C03618=1103.149,283.169,-77.538,179.285,15.809,151.491
C03619=1103.143,282.921,-77.509,179.281,15.808,151.491
C03620=1103.138,282.672,-77.480,179.278,15.807,151.492
C03621=1103.132,282.424,-77.450,179.274,15.805,151.492
C03622=1103.126,282.176,-77.422,179.271,15.805,151.493
C03623=1103.121,281.927,-77.393,179.267,15.803,151.493
C03624=1103.115,281.679,-77.364,179.264,15.802,151.494
C03625=1103.109,281.431,-77.334,179.260,15.801,151.494
C03626=1103.104,281.183,-77.305,179.256,15.800,151.495
C03627=1103.098,280.935,-77.276,179.252,15.799,151.495
C03628=1103.092,280.687,-77.247,179.249,15.798,151.496
C03629=1103.087,280.438,-77.218,179.245,15.797,151.496
C03630=1103.081,280.190,-77.189,179.242,15.796,151.497
C03631=1103.076,279.942,-77.159,179.238,15.795,151.497
C03632=1103.069,279.694,-77.130,179.235,15.794,151.498
C03633=1103.064,279.446,-77.101,179.231,15.793,151.498
C03634=1103.059,279.197,-77.073,179.227,15.792,151.499
C03635=1103.053,278.949,-77.043,179.224,15.791,151.499
C03636=1103.047,278.701,-77.014,179.220,15.790,151.500
C03637=1103.041,278.453,-76.986,179.216,15.789,151.500
C03638=1103.036,278.204,-76.956,179.212,15.788,151.501
C03639=1103.030,277.956,-76.927,179.209,15.787,151.502
C03640=1103.025,277.708,-76.899,179.205,15.786,151.502
C03641=1103.019,277.460,-76.870,179.202,15.785,151.503
C03642=1103.013,277.211,-76.841,179.198,15.784,151.503
C03643=1103.008,276.963,-76.812,179.195,15.783,151.504
C03644=1103.000,276.606,-76.771,179.189,15.782,151.504
C03645=1102.991,276.250,-76.729,179.184,15.781,151.505
C03646=1102.984,275.893,-76.688,179.179,15.780,151.506
C03647=1102.975,275.536,-76.647,179.174,15.778,151.507
C03648=1102.969,275.288,-76.618,179.170,15.777,151.507
C03649=1102.964,275.039,-76.589,179.167,15.776,151.508
C03650=1102.958,274.791,-76.560,179.163,15.775,151.508
C03651=1102.952,274.543,-76.532,179.159,15.774,151.509
C03652=1102.946,274.294,-76.503,179.155,15.773,151.509
C03653=1102.941,274.046,-76.474,179.152,15.772,151.510
C03654=1102.935,273.797,-76.446,179.148,15.771,151.511
C03655=1102.930,273.550,-76.417,179.145,15.770,151.511
C03656=1102.924,273.301,-76.389,179.141,15.769,151.512
C03657=1102.918,273.053,-76.359,179.138,15.769,151.512
C03658=1102.913,272.805,-76.331,179.134,15.767,151.513
C03659=1102.907,272.556,-76.303,179.130,15.767,151.513
C03660=1102.901,272.308,-76.274,179.127,15.766,151.514
C03661=1102.896,272.060,-76.246,179.123,15.765,151.515
C03662=1102.891,271.811,-76.217,179.120,15.764,151.515
C03663=1102.885,271.563,-76.188,179.116,15.763,151.516
C03664=1102.879,271.314,-76.160,179.112,15.762,151.516
C03665=1102.873,271.066,-76.132,179.108,15.762,151.517
C03666=1102.867,270.818,-76.103,179.105,15.761,151.517
C03667=1102.862,270.570,-76.075,179.101,15.760,151.518
C03668=1102.856,270.321,-76.047,179.098,15.759,151.518
C03669=1102.851,270.073,-76.019,179.094,15.758,151.519
C03670=1102.845,269.825,-75.989,179.090,15.757,151.520
C03671=1102.840,269.577,-75.961,179.086,15.756,151.520
C03672=1102.834,269.328,-75.933,179.083,15.756,151.521
C03673=1102.828,269.079,-75.904,179.080,15.755,151.521
C03674=1102.822,268.831,-75.876,179.076,15.754,151.522
C03675=1102.816,268.583,-75.848,179.072,15.753,151.522
C03676=1102.811,268.335,-75.819,179.068,15.752,151.523
C03677=1102.805,268.086,-75.791,179.065,15.751,151.524
C03678=1102.800,267.838,-75.763,179.061,15.750,151.524
C03679=1102.794,267.590,-75.735,179.057,15.750,151.525
C03680=1102.788,267.342,-75.707,179.054,15.749,151.525
C03681=1102.782,267.093,-75.679,179.050,15.748,151.526
C03682=1102.777,266.845,-75.651,179.047,15.748,151.527
C03683=1102.771,266.596,-75.622,179.043,15.746,151.527
C03684=1102.766,266.348,-75.594,179.040,15.746,151.528
C03685=1102.760,266.100,-75.566,179.035,15.745,151.528
C03686=1102.754,265.851,-75.538,179.032,15.744,151.529
C03687=1102.749,265.603,-75.510,179.028,15.743,151.529
C03688=1102.743,265.354,-75.482,179.025,15.743,151.530
C03689=1102.738,265.106,-75.454,179.021,15.742,151.531
C03690=1102.732,264.858,-75.425,179.017,15.741,151.531
C03691=1102.726,264.610,-75.398,179.014,15.740,151.532
C03692=1102.720,264.362,-75.370,179.010,15.739,151.532
C03693=1102.714,264.113,-75.342,179.006,15.739,151.533
C03694=1102.709,263.865,-75.314,179.003,15.738,151.534
C03695=1102.703,263.616,-75.286,178.999,15.737,151.534
C03696=1102.695,263.263,-75.246,178.994,15.736,151.535
C03697=1102.686,262.908,-75.207,178.988,15.735,151.536
C03698=1102.679,262.554,-75.167,178.984,15.735,151.537
C03699=1102.670,262.200,-75.127,178.978,15.733,151.538
C03700=1102.665,261.952,-75.099,178.974,15.732,151.538
C03701=1102.659,261.703,-75.071,178.971,15.732,151.539
C03702=1102.653,261.455,-75.044,178.968,15.731,151.539
C03703=1102.647,261.206,-75.016,178.963,15.730,151.540
C03704=1102.642,260.958,-74.988,178.960,15.730,151.541
C03705=1102.636,260.710,-74.960,178.956,15.729,151.541
C03706=1102.630,260.461,-74.933,178.953,15.728,151.542
C03707=1102.625,260.213,-74.905,178.949,15.728,151.543
C03708=1102.618,259.964,-74.877,178.945,15.727,151.543
C03709=1102.613,259.716,-74.850,178.941,15.726,151.544
C03710=1102.608,259.468,-74.822,178.938,15.726,151.544
C03711=1102.601,259.219,-74.794,178.934,15.725,151.545
C03712=1102.596,258.971,-74.767,178.931,15.724,151.546
C03713=1102.591,258.723,-74.739,178.926,15.723,151.546
C03714=1102.584,258.474,-74.711,178.923,15.723,151.547
C03715=1102.579,258.225,-74.684,178.920,15.722,151.548
C03716=1102.573,257.977,-74.656,178.915,15.721,151.548
C03717=1102.567,257.728,-74.629,178.912,15.721,151.549
C03718=1102.562,257.480,-74.601,178.909,15.721,151.549
C03719=1102.556,257.233,-74.574,178.905,15.719,151.550
C03720=1102.550,256.983,-74.546,178.901,15.719,151.551
C03721=1102.545,256.735,-74.518,178.898,15.718,151.551
C03722=1102.539,256.487,-74.491,178.894,15.717,151.552
C03723=1102.533,256.238,-74.463,178.890,15.717,151.552
C03724=1102.527,255.990,-74.436,178.886,15.716,151.553
C03725=1102.522,255.742,-74.409,178.883,15.715,151.554
C03726=1102.517,255.493,-74.381,178.879,15.715,151.554
C03727=1102.510,255.244,-74.354,178.875,15.714,151.555
C03728=1102.505,254.996,-74.326,178.872,15.714,151.556
C03729=1102.499,254.747,-74.300,178.868,15.713,151.556
C03730=1102.494,254.499,-74.272,178.864,15.712,151.557
C03731=1102.488,254.250,-74.245,178.861,15.712,151.558
C03732=1102.483,254.002,-74.217,178.858,15.711,151.558
C03733=1102.476,253.754,-74.190,178.853,15.710,151.559
C03734=1102.471,253.505,-74.163,178.850,15.710,151.559
C03735=1102.465,253.257,-74.135,178.847,15.709,151.560
C03736=1102.460,253.008,-74.108,178.843,15.708,151.561
C03737=1102.454,252.760,-74.081,178.839,15.708,151.561
C03738=1102.449,252.511,-74.054,178.835,15.707,151.562
C03739=1102.443,252.263,-74.027,178.832,15.706,151.562
C03740=1102.438,252.015,-73.999,178.828,15.706,151.563
C03741=1102.431,251.766,-73.972,178.824,15.705,151.564
C03742=1102.426,251.517,-73.945,178.821,15.705,151.564
C03743=1102.420,251.269,-73.918,178.817,15.704,151.565
C03744=1102.415,251.021,-73.891,178.813,15.703,151.566
C03745=1102.410,250.772,-73.864,178.810,15.702,151.566
C03746=1102.404,250.524,-73.837,178.806,15.702,151.567
C03747=1102.398,250.274,-73.810,178.802,15.701,151.568
C03748=1102.390,249.918,-73.770,178.797,15.701,151.568
C03749=1102.382,249.561,-73.732,178.792,15.700,151.569
C03750=1102.374,249.204,-73.693,178.787,15.699,151.570
C03751=1102.366,248.847,-73.653,178.781,15.698,151.571
C03752=1102.361,248.599,-73.627,178.778,15.697,151.572
C03753=1102.355,248.351,-73.600,178.775,15.697,151.572
C03754=1102.350,248.102,-73.573,178.770,15.696,151.573
C03755=1102.344,247.854,-73.546,178.767,15.695,151.574
C03756=1102.339,247.605,-73.519,178.764,15.695,151.574
C03757=1102.333,247.357,-73.492,178.760,15.694,151.575
C03758=1102.327,247.108,-73.466,178.756,15.694,151.575
C03759=1102.322,246.860,-73.439,178.753,15.693,151.576
C03760=1102.317,246.611,-73.412,178.749,15.692,151.577
C03761=1102.311,246.363,-73.385,178.745,15.692,151.577
C03762=1102.304,246.114,-73.358,178.741,15.692,151.578
C03763=1102.299,245.865,-73.332,178.738,15.691,151.579
C03764=1102.294,245.617,-73.304,178.734,15.690,151.579
C03765=1102.288,245.368,-73.278,178.730,15.690,151.580
C03766=1102.282,245.120,-73.251,178.727,15.689,151.581
C03767=1102.276,244.872,-73.224,178.723,15.688,151.581
C03768=1102.272,244.622,-73.198,178.719,15.688,151.582
C03769=1102.266,244.374,-73.171,178.716,15.688,151.583
C03770=1102.260,244.126,-73.145,178.713,15.687,151.583
C03771=1102.254,243.877,-73.118,178.708,15.687,151.584
C03772=1102.248,243.629,-73.091,178.705,15.686,151.584
C03773=1102.243,243.381,-73.065,178.702,15.686,151.585
C03774=1102.238,243.131,-73.038,178.697,15.685,151.586
C03775=1102.232,242.883,-73.011,178.694,15.684,151.586
C03776=1102.226,242.635,-72.985,178.691,15.684,151.587
C03777=1102.221,242.386,-72.958,178.687,15.684,151.588
C03778=1102.215,242.138,-72.931,178.683,15.683,151.589
C03779=1102.209,241.889,-72.906,178.680,15.682,151.589
C03780=1102.204,241.641,-72.879,178.676,15.682,151.590
C03781=1102.198,241.392,-72.852,178.672,15.681,151.590
C03782=1102.192,241.144,-72.826,178.668,15.681,151.591
C03783=1102.187,240.895,-72.800,178.665,15.681,151.592
C03784=1102.181,240.646,-72.773,178.661,15.680,151.592
C03785=1102.175,240.398,-72.746,178.657,15.679,151.593
C03786=1102.170,240.149,-72.720,178.654,15.679,151.594
C03787=1102.164,239.901,-72.694,178.650,15.679,151.595
C03788=1102.158,239.652,-72.667,178.647,15.678,151.595
C03789=1102.153,239.403,-72.641,178.642,15.677,151.596
C03790=1102.147,239.155,-72.615,178.639,15.677,151.597
C03791=1102.141,238.906,-72.589,178.635,15.677,151.597
C03792=1102.136,238.658,-72.562,178.632,15.676,151.598
C03793=1102.130,238.409,-72.535,178.628,15.676,151.598
C03794=1102.124,238.160,-72.509,178.624,15.675,151.599
C03795=1102.119,237.912,-72.483,178.621,15.675,151.600
C03796=1102.113,237.663,-72.457,178.617,15.675,151.601
C03797=1102.107,237.415,-72.431,178.613,15.674,151.601
C03798=1102.101,237.166,-72.405,178.610,15.674,151.602
C03799=1102.095,236.918,-72.378,178.606,15.673,151.603
C03800=1102.088,236.554,-72.340,178.601,15.672,151.603
C03801=1102.079,236.190,-72.302,178.595,15.672,151.604
C03802=1102.071,235.827,-72.263,178.591,15.671,151.605
C03803=1102.063,235.463,-72.226,178.585,15.671,151.606
C03804=1102.057,235.214,-72.199,178.581,15.670,151.607
C03805=1102.052,234.965,-72.173,178.578,15.670,151.608
C03806=1102.046,234.718,-72.147,178.574,15.669,151.608
C03807=1102.041,234.469,-72.121,178.570,15.669,151.609
C03808=1102.035,234.220,-72.095,178.567,15.669,151.610
C03809=1102.029,233.972,-72.069,178.563,15.668,151.610
C03810=1102.023,233.723,-72.043,178.559,15.667,151.611
C03811=1102.018,233.474,-72.017,178.556,15.667,151.612
C03812=1102.013,233.226,-71.991,178.552,15.667,151.612
C03813=1102.007,232.977,-71.966,178.549,15.667,151.613
C03814=1102.001,232.728,-71.940,178.545,15.666,151.614
C03815=1101.996,232.479,-71.914,178.541,15.666,151.615
C03816=1101.990,232.231,-71.887,178.538,15.665,151.615
C03817=1101.984,231.982,-71.862,178.534,15.665,151.616
C03818=1101.979,231.734,-71.836,178.530,15.665,151.617
C03819=1101.973,231.485,-71.810,178.526,15.664,151.617
C03820=1101.968,231.237,-71.784,178.523,15.663,151.618
C03821=1101.961,230.988,-71.758,178.519,15.663,151.619
C03822=1101.956,230.739,-71.732,178.516,15.663,151.619
C03823=1101.951,230.491,-71.707,178.512,15.662,151.620
C03824=1101.945,230.242,-71.681,178.508,15.662,151.621
C03825=1101.939,229.993,-71.655,178.505,15.661,151.621
C03826=1101.933,229.745,-71.629,178.501,15.661,151.622
C03827=1101.927,229.496,-71.603,178.497,15.661,151.623
C03828=1101.923,229.248,-71.578,178.494,15.661,151.623
C03829=1101.916,228.999,-71.553,178.491,15.660,151.624
C03830=1101.911,228.750,-71.527,178.486,15.659,151.625
C03831=1101.905,228.502,-71.501,178.483,15.659,151.625
C03832=1101.900,228.253,-71.476,178.479,15.659,151.626
C03833=1101.894,228.005,-71.450,178.476,15.659,151.627
C03834=1101.888,227.756,-71.424,178.472,15.659,151.628
C03835=1101.882,227.507,-71.399,178.468,15.658,151.628
C03836=1101.877,227.259,-71.374,178.464,15.658,151.629
C03837=1101.872,227.010,-71.348,178.461,15.658,151.630
C03838=1101.865,226.761,-71.322,178.458,15.657,151.630
C03839=1101.860,226.512,-71.296,178.454,15.657,151.631
C03840=1101.854,226.264,-71.271,178.451,15.657,151.632
C03841=1101.849,226.015,-71.245,178.446,15.656,151.632
C03842=1101.843,225.766,-71.220,178.443,15.656,151.633
C03843=1101.838,225.518,-71.194,178.439,15.655,151.634
C03844=1101.832,225.269,-71.169,178.436,15.655,151.635
C03845=1101.826,225.020,-71.143,178.432,15.655,151.635
C03846=1101.820,224.772,-71.118,178.429,15.654,151.636
C03847=1101.815,224.523,-71.094,178.425,15.654,151.636
C03848=1101.809,224.274,-71.068,178.421,15.653,151.637
C03849=1101.803,224.026,-71.042,178.417,15.653,151.638
C03850=1101.798,223.777,-71.017,178.414,15.653,151.639
C03851=1101.792,223.529,-70.991,178.410,15.653,151.639
C03852=1101.784,223.156,-70.954,178.405,15.652,151.640
C03853=1101.776,222.784,-70.916,178.399,15.651,151.641
C03854=1101.767,222.412,-70.878,178.394,15.651,151.642
C03855=1101.759,222.040,-70.840,178.389,15.651,151.643
C03856=1101.753,221.792,-70.815,178.385,15.651,151.644
C03857=1101.747,221.543,-70.790,178.382,15.650,151.645
C03858=1101.741,221.294,-70.764,178.377,15.650,151.646
C03859=1101.737,221.045,-70.740,178.374,15.649,151.646
C03860=1101.730,220.797,-70.714,178.370,15.649,151.647
C03861=1101.724,220.548,-70.689,178.367,15.649,151.648
C03862=1101.719,220.299,-70.665,178.363,15.649,151.648
C03863=1101.713,220.050,-70.639,178.360,15.649,151.649
C03864=1101.707,219.802,-70.613,178.356,15.649,151.650
C03865=1101.702,219.553,-70.589,178.352,15.648,151.651
C03866=1101.696,219.304,-70.564,178.349,15.647,151.651
C03867=1101.691,219.056,-70.539,178.345,15.647,151.652
C03868=1101.685,218.807,-70.514,178.341,15.647,151.653
C03869=1101.679,218.559,-70.489,178.338,15.647,151.653
C03870=1101.673,218.310,-70.464,178.334,15.647,151.654
C03871=1101.668,218.061,-70.438,178.331,15.646,151.655
C03872=1101.663,217.812,-70.414,178.327,15.646,151.655
C03873=1101.656,217.563,-70.388,178.323,15.645,151.656
C03874=1101.651,217.315,-70.364,178.319,15.645,151.657
C03875=1101.645,217.066,-70.339,178.316,15.645,151.658
C03876=1101.640,216.817,-70.314,178.312,15.645,151.658
C03877=1101.634,216.569,-70.289,178.309,15.645,151.659
C03878=1101.629,216.320,-70.264,178.305,15.645,151.660
C03879=1101.623,216.071,-70.239,178.302,15.644,151.660
C03880=1101.617,215.823,-70.215,178.298,15.644,151.661
C03881=1101.611,215.574,-70.189,178.295,15.644,151.662
C03882=1101.606,215.326,-70.165,178.291,15.643,151.662
C03883=1101.601,215.076,-70.140,178.287,15.643,151.663
C03884=1101.595,214.828,-70.115,178.284,15.643,151.664
C03885=1101.589,214.579,-70.090,178.280,15.642,151.665
C03886=1101.584,214.331,-70.065,178.276,15.642,151.665
C03887=1101.578,214.081,-70.041,178.273,15.642,151.666
C03888=1101.572,213.833,-70.017,178.269,15.642,151.667
C03889=1101.567,213.585,-69.992,178.266,15.642,151.667
C03890=1101.561,213.336,-69.967,178.262,15.642,151.668
C03891=1101.556,213.087,-69.943,178.258,15.641,151.669
C03892=1101.550,212.838,-69.918,178.254,15.641,151.670
C03893=1101.544,212.590,-69.893,178.251,15.641,151.670
C03894=1101.538,212.340,-69.869,178.247,15.640,151.671
C03895=1101.533,212.092,-69.844,178.244,15.640,151.672
C03896=1101.527,211.843,-69.819,178.240,15.640,151.672
C03897=1101.521,211.595,-69.795,178.237,15.640,151.673
C03898=1101.516,211.346,-69.770,178.233,15.640,151.674
C03899=1101.510,211.097,-69.746,178.230,15.639,151.674
C03900=1101.505,210.848,-69.722,178.226,15.639,151.675
C03901=1101.499,210.599,-69.696,178.223,15.639,151.676
C03902=1101.493,210.351,-69.672,178.218,15.638,151.677
C03903=1101.487,210.102,-69.647,178.215,15.638,151.677
C03904=1101.480,209.733,-69.611,178.210,15.638,151.678
C03905=1101.471,209.366,-69.575,178.204,15.637,151.679
C03906=1101.463,208.997,-69.539,178.199,15.638,151.680
C03907=1101.455,208.628,-69.503,178.194,15.637,151.682
C03908=1101.431,207.624,-69.405,178.158,15.629,151.687
C03909=1101.426,207.375,-69.381,178.154,15.629,151.688
C03910=1101.420,207.126,-69.356,178.150,15.630,151.689
C03911=1101.414,206.878,-69.332,178.146,15.630,151.690
C03912=1101.409,206.629,-69.308,178.143,15.631,151.691
C03913=1101.403,206.380,-69.283,178.139,15.632,151.692
C03914=1101.397,206.132,-69.260,178.135,15.632,151.693
C03915=1101.392,205.882,-69.236,178.131,15.633,151.694
C03916=1101.387,205.634,-69.212,178.128,15.634,151.695
C03917=1101.381,205.384,-69.187,178.124,15.634,151.696
C03918=1101.375,205.136,-69.164,178.120,15.635,151.697
C03919=1101.369,204.888,-69.139,178.116,15.635,151.698
C03920=1101.363,204.638,-69.115,178.112,15.636,151.699
C03921=1101.357,204.390,-69.091,178.109,15.637,151.700
C03922=1101.352,204.141,-69.068,178.105,15.637,151.700
C03923=1101.347,203.892,-69.043,178.100,15.638,151.701
C03924=1101.340,203.643,-69.019,178.097,15.638,151.702
C03925=1101.335,203.395,-68.995,178.094,15.639,151.703
C03926=1101.330,203.145,-68.972,178.089,15.640,151.704
C03927=1101.324,202.897,-68.948,178.086,15.640,151.705
C03928=1101.319,202.649,-68.924,178.082,15.641,151.706
C03929=1101.312,202.400,-68.900,178.077,15.641,151.707
C03930=1101.307,202.150,-68.876,178.074,15.642,151.708
C03931=1101.301,201.902,-68.852,178.070,15.643,151.709
C03932=1101.295,201.653,-68.828,178.066,15.643,151.710
C03933=1101.289,201.405,-68.804,178.063,15.644,151.711
C03934=1101.284,201.155,-68.781,178.059,15.645,151.712
C03935=1101.278,200.907,-68.757,178.055,15.645,151.713
C03936=1101.272,200.658,-68.732,178.051,15.646,151.714
C03937=1101.267,200.409,-68.709,178.047,15.646,151.715
C03938=1101.260,200.161,-68.686,178.044,15.647,151.715
C03939=1101.255,199.911,-68.662,178.040,15.648,151.717
C03940=1101.249,199.662,-68.638,178.036,15.649,151.717
C03941=1101.244,199.414,-68.614,178.032,15.649,151.718
C03942=1101.238,199.165,-68.591,178.029,15.650,151.719
C03943=1101.233,198.916,-68.567,178.025,15.651,151.720
C03944=1101.227,198.668,-68.544,178.021,15.651,151.721
C03945=1101.220,198.419,-68.520,178.017,15.652,151.722
C03946=1101.215,198.169,-68.496,178.014,15.653,151.723
C03947=1101.209,197.921,-68.473,178.010,15.653,151.724
C03948=1101.204,197.672,-68.449,178.006,15.654,151.725
C03949=1101.198,197.424,-68.425,178.002,15.654,151.726
C03950=1101.192,197.175,-68.402,177.999,15.655,151.727
C03951=1101.187,196.926,-68.378,177.995,15.656,151.728
C03952=1101.181,196.676,-68.355,177.991,15.656,151.729
C03953=1101.175,196.428,-68.331,177.987,15.656,151.729
C03954=1101.170,196.179,-68.308,177.984,15.657,151.730
C03955=1101.164,195.931,-68.284,177.980,15.658,151.731
C03956=1101.159,195.682,-68.260,177.976,15.658,151.732
C03957=1101.153,195.433,-68.237,177.972,15.659,151.733
C03958=1101.147,195.184,-68.214,177.969,15.660,151.734
C03959=1101.142,194.935,-68.190,177.965,15.660,151.735
C03960=1101.135,194.686,-68.166,177.961,15.661,151.736
C03961=1101.130,194.437,-68.143,177.957,15.661,151.737
C03962=1101.124,194.188,-68.120,177.954,15.662,151.738
C03963=1101.119,193.940,-68.096,177.950,15.662,151.739
C03964=1101.113,193.691,-68.073,177.946,15.663,151.739
C03965=1101.107,193.442,-68.050,177.942,15.663,151.741
C03966=1101.102,193.193,-68.026,177.939,15.664,151.741
C03967=1101.096,192.944,-68.003,177.935,15.665,151.742
C03968=1101.090,192.696,-67.980,177.931,15.665,151.743
C03969=1101.084,192.423,-67.954,177.927,15.666,151.744
C03970=1101.079,192.150,-67.929,177.923,15.666,151.745
C03971=1101.071,191.877,-67.903,177.919,15.667,151.746
C03972=1101.066,191.604,-67.878,177.915,15.667,151.747
C03973=1101.059,191.356,-67.854,177.911,15.668,151.748
C03974=1101.054,191.107,-67.831,177.908,15.669,151.749
C03975=1101.049,190.858,-67.808,177.904,15.669,151.750
C03976=1101.043,190.609,-67.785,177.900,15.670,151.751
C03977=1101.037,190.360,-67.762,177.896,15.670,151.752
C03978=1101.032,190.112,-67.738,177.893,15.671,151.753
C03979=1101.026,189.863,-67.715,177.889,15.671,151.753
C03980=1101.021,189.614,-67.692,177.886,15.672,151.754
C03981=1101.015,189.365,-67.669,177.882,15.672,151.755
C03982=1101.010,189.116,-67.645,177.879,15.673,151.756
C03983=1101.005,188.868,-67.623,177.875,15.673,151.757
C03984=1100.999,188.619,-67.600,177.871,15.674,151.758
C03985=1100.993,188.370,-67.577,177.867,15.674,151.759
C03986=1100.987,188.121,-67.554,177.864,15.675,151.760
C03987=1100.982,187.872,-67.531,177.860,15.675,151.760
C03988=1100.977,187.623,-67.507,177.856,15.676,151.761
C03989=1100.971,187.374,-67.484,177.852,15.676,151.762
C03990=1100.965,187.125,-67.461,177.849,15.677,151.763
C03991=1100.959,186.877,-67.438,177.845,15.677,151.764
C03992=1100.954,186.627,-67.415,177.841,15.678,151.765
C03993=1100.948,186.378,-67.393,177.838,15.677,151.766
C03994=1100.943,186.129,-67.369,177.835,15.678,151.766
C03995=1100.938,185.881,-67.346,177.831,15.679,151.767
C03996=1100.932,185.632,-67.323,177.827,15.679,151.768
C03997=1100.927,185.383,-67.301,177.824,15.680,151.769
C03998=1100.921,185.134,-67.278,177.820,15.680,151.770
C03999=1100.915,184.885,-67.255,177.816,15.681,151.771
C04000=1100.909,184.636,-67.232,177.812,15.681,151.772
C04001=1100.904,184.387,-67.209,177.809,15.682,151.773
C04002=1100.898,184.139,-67.186,177.805,15.682,151.774
C04003=1100.891,183.890,-67.163,177.802,15.683,151.774
C04004=1100.886,183.641,-67.141,177.799,15.684,151.775
C04005=1100.880,183.392,-67.118,177.795,15.684,151.776
C04006=1100.875,183.143,-67.095,177.791,15.684,151.777
C04007=1100.869,182.894,-67.072,177.787,15.685,151.778
C04008=1100.863,182.645,-67.049,177.784,15.686,151.779
C04009=1100.857,182.396,-67.027,177.780,15.686,151.780
C04010=1100.851,182.147,-67.004,177.776,15.687,151.781
C04011=1100.846,181.899,-66.982,177.773,15.688,151.781
C04012=1100.840,181.650,-66.959,177.769,15.688,151.782
C04013=1100.835,181.401,-66.936,177.765,15.688,151.783
C04014=1100.829,181.152,-66.913,177.761,15.689,151.784
C04015=1100.822,180.903,-66.891,177.758,15.690,151.785
C04016=1100.817,180.654,-66.869,177.754,15.690,151.786
C04017=1100.811,180.405,-66.846,177.751,15.690,151.787
C04018=1100.805,180.156,-66.823,177.748,15.691,151.788
C04019=1100.799,179.907,-66.801,177.744,15.692,151.789
C04020=1100.794,179.659,-66.779,177.740,15.692,151.789
C04021=1100.788,179.410,-66.756,177.737,15.693,151.790
C04022=1100.783,179.161,-66.733,177.733,15.693,151.791
C04023=1100.777,178.912,-66.711,177.729,15.693,151.792
C04024=1100.771,178.663,-66.688,177.725,15.694,151.793
C04025=1100.765,178.414,-66.665,177.722,15.695,151.794
C04026=1100.760,178.164,-66.643,177.718,15.695,151.795
C04027=1100.754,177.916,-66.621,177.715,15.695,151.796
C04028=1100.748,177.667,-66.599,177.712,15.696,151.796
C04029=1100.743,177.418,-66.576,177.708,15.696,151.797
C04030=1100.737,177.169,-66.553,177.704,15.697,151.798
C04031=1100.731,176.920,-66.531,177.701,15.698,151.799
C04032=1100.726,176.672,-66.509,177.697,15.698,151.800
C04033=1100.719,176.399,-66.484,177.693,15.698,151.801
C04034=1100.712,176.125,-66.460,177.689,15.699,151.802
C04035=1100.707,175.852,-66.435,177.686,15.699,151.802
C04036=1100.701,175.579,-66.411,177.681,15.700,151.803
C04037=1100.695,175.331,-66.389,177.678,15.700,151.804
C04038=1100.689,175.081,-66.366,177.675,15.701,151.805
C04039=1100.684,174.832,-66.344,177.671,15.701,151.806
C04040=1100.677,174.583,-66.322,177.667,15.702,151.807
C04041=1100.672,174.335,-66.299,177.664,15.702,151.808
C04042=1100.667,174.085,-66.277,177.660,15.702,151.808
C04043=1100.661,173.836,-66.255,177.656,15.703,151.809
C04044=1100.655,173.587,-66.232,177.653,15.703,151.810
C04045=1100.650,173.338,-66.211,177.650,15.704,151.811
C04046=1100.644,173.090,-66.188,177.646,15.704,151.812
C04047=1100.638,172.840,-66.166,177.642,15.704,151.813
C04048=1100.633,172.592,-66.144,177.639,15.705,151.813
C04049=1100.627,172.343,-66.122,177.635,15.705,151.814
C04050=1100.622,172.093,-66.100,177.632,15.705,151.815
C04051=1100.616,171.846,-66.078,177.629,15.706,151.816
C04052=1100.610,171.596,-66.055,177.625,15.706,151.817
C04053=1100.605,171.347,-66.033,177.621,15.707,151.818
C04054=1100.599,171.098,-66.012,177.618,15.708,151.818
C04055=1100.594,170.849,-65.989,177.615,15.708,151.819
C04056=1100.587,170.600,-65.967,177.611,15.708,151.820
C04057=1100.583,170.351,-65.945,177.607,15.708,151.821
C04058=1100.577,170.102,-65.922,177.604,15.709,151.822
C04059=1100.571,169.853,-65.901,177.601,15.709,151.822
C04060=1100.566,169.604,-65.879,177.597,15.709,151.823
C04061=1100.560,169.355,-65.857,177.594,15.710,151.824
C04062=1100.555,169.107,-65.835,177.590,15.710,151.825
C04063=1100.548,168.858,-65.813,177.587,15.710,151.826
C04064=1100.543,168.608,-65.791,177.583,15.711,151.827
C04065=1100.537,168.360,-65.770,177.580,15.711,151.827
C04066=1100.532,168.110,-65.747,177.576,15.711,151.828
C04067=1100.526,167.862,-65.726,177.573,15.712,151.829
C04068=1100.521,167.613,-65.703,177.569,15.712,151.830
C04069=1100.515,167.363,-65.681,177.566,15.712,151.830
C04070=1100.510,167.115,-65.660,177.563,15.713,151.831
C04071=1100.504,166.865,-65.637,177.559,15.713,151.832
C04072=1100.499,166.617,-65.616,177.555,15.714,151.833
C04073=1100.493,166.367,-65.594,177.552,15.714,151.834
C04074=1100.488,166.119,-65.573,177.549,15.714,151.834
C04075=1100.482,165.869,-65.550,177.545,15.714,151.835
C04076=1100.477,165.621,-65.529,177.542,15.714,151.836
C04077=1100.471,165.371,-65.508,177.539,15.715,151.837
C04078=1100.465,165.123,-65.485,177.535,15.715,151.838
C04079=1100.459,164.874,-65.463,177.531,15.715,151.838
C04080=1100.454,164.625,-65.441,177.528,15.716,151.839
C04081=1100.448,164.376,-65.420,177.525,15.716,151.840
C04082=1100.443,164.127,-65.398,177.521,15.716,151.841
C04083=1100.437,163.878,-65.376,177.518,15.717,151.842
C04084=1100.433,163.628,-65.355,177.514,15.717,151.842
C04085=1100.427,163.379,-65.334,177.511,15.717,151.843
C04086=1100.422,163.130,-65.312,177.508,15.718,151.844
C04087=1100.416,162.881,-65.290,177.504,15.718,151.845
C04088=1100.410,162.633,-65.269,177.501,15.718,151.845
C04089=1100.405,162.383,-65.247,177.498,15.719,151.846
C04090=1100.399,162.135,-65.225,177.494,15.719,151.847
C04091=1100.394,161.885,-65.203,177.490,15.719,151.848
C04092=1100.388,161.637,-65.182,177.488,15.719,151.848
C04093=1100.382,161.388,-65.160,177.484,15.719,151.849
C04094=1100.376,161.139,-65.139,177.480,15.720,151.850
C04095=1100.371,160.889,-65.117,177.477,15.720,151.851
C04096=1100.366,160.640,-65.096,177.474,15.720,151.852
C04097=1100.359,160.367,-65.072,177.470,15.721,151.852
C04098=1100.353,160.094,-65.049,177.466,15.721,151.853
C04099=1100.347,159.820,-65.025,177.462,15.722,151.854
C04100=1100.341,159.547,-65.002,177.459,15.721,151.855
C04101=1100.335,159.298,-64.980,177.456,15.723,151.856
C04102=1100.329,159.049,-64.959,177.452,15.722,151.857
C04103=1100.324,158.800,-64.938,177.448,15.722,151.857
C04104=1100.318,158.550,-64.916,177.445,15.723,151.858
C04105=1100.313,158.302,-64.895,177.442,15.723,151.859
C04106=1100.307,158.053,-64.873,177.438,15.723,151.860
C04107=1100.301,157.804,-64.853,177.435,15.724,151.860
C04108=1100.295,157.554,-64.831,177.432,15.724,151.861
C04109=1100.290,157.306,-64.810,177.428,15.724,151.862
C04110=1100.283,157.057,-64.788,177.425,15.725,151.863
C04111=1100.279,156.807,-64.767,177.422,15.725,151.863
C04112=1100.273,156.559,-64.746,177.418,15.725,151.864
C04113=1100.267,156.309,-64.724,177.415,15.726,151.865
C04114=1100.262,156.060,-64.703,177.411,15.726,151.866
C04115=1100.256,155.811,-64.682,177.408,15.726,151.867
C04116=1100.250,155.563,-64.660,177.405,15.726,151.867
C04117=1100.245,155.314,-64.640,177.402,15.726,151.868
C04118=1100.239,155.064,-64.618,177.398,15.727,151.869
C04119=1100.233,154.815,-64.598,177.395,15.727,151.870
C04120=1100.227,154.566,-64.576,177.391,15.727,151.870
C04121=1100.222,154.317,-64.555,177.389,15.728,151.871
C04122=1100.217,154.068,-64.534,177.385,15.728,151.872
C04123=1100.210,153.819,-64.513,177.381,15.728,151.873
C04124=1100.205,153.570,-64.492,177.379,15.728,151.873
C04125=1100.199,153.321,-64.470,177.375,15.729,151.874
C04126=1100.194,153.072,-64.450,177.371,15.729,151.875
C04127=1100.188,152.823,-64.429,177.368,15.729,151.876
C04128=1100.182,152.573,-64.408,177.365,15.729,151.876
C04129=1100.177,152.325,-64.386,177.361,15.729,151.877
C04130=1100.171,152.076,-64.366,177.359,15.730,151.878
C04131=1100.165,151.827,-64.344,177.355,15.730,151.879
C04132=1100.160,151.577,-64.324,177.352,15.730,151.879
C04133=1100.154,151.329,-64.302,177.349,15.730,151.880
C04134=1100.149,151.079,-64.282,177.345,15.730,151.881
C04135=1100.143,150.831,-64.260,177.342,15.731,151.881
C04136=1100.138,150.581,-64.240,177.339,15.731,151.882
C04137=1100.132,150.332,-64.218,177.335,15.731,151.883
C04138=1100.126,150.083,-64.197,177.332,15.731,151.884
C04139=1100.121,149.834,-64.177,177.329,15.731,151.884
C04140=1100.115,149.586,-64.156,177.325,15.731,151.885
C04141=1100.109,149.336,-64.135,177.322,15.732,151.886
C04142=1100.103,149.087,-64.114,177.319,15.732,151.887
C04143=1100.098,148.838,-64.094,177.316,15.732,151.887
C04144=1100.092,148.589,-64.073,177.313,15.732,151.888
C04145=1100.087,148.340,-64.051,177.309,15.732,151.889
C04146=1100.081,148.091,-64.031,177.306,15.733,151.889
C04147=1100.075,147.841,-64.010,177.303,15.733,151.890
C04148=1100.069,147.593,-63.989,177.299,15.733,151.891
C04149=1100.064,147.344,-63.969,177.296,15.733,151.892
C04150=1100.059,147.095,-63.948,177.293,15.733,151.892
C04151=1100.053,146.845,-63.927,177.289,15.733,151.893
C04152=1100.047,146.597,-63.906,177.286,15.734,151.894
C04153=1100.041,146.347,-63.886,177.283,15.734,151.895
C04154=1100.036,146.098,-63.865,177.280,15.735,151.895
C04155=1100.030,145.849,-63.844,177.276,15.735,151.896
C04156=1100.024,145.600,-63.824,177.273,15.734,151.897
C04157=1100.019,145.351,-63.803,177.270,15.735,151.898
C04158=1100.013,145.102,-63.783,177.266,15.735,151.898
C04159=1100.008,144.852,-63.762,177.263,15.735,151.899
C04160=1100.002,144.603,-63.742,177.260,15.735,151.900
C04161=1099.996,144.330,-63.718,177.257,15.736,151.900
C04162=1099.989,144.056,-63.696,177.253,15.736,151.901
C04163=1099.983,143.783,-63.674,177.249,15.736,151.902
C04164=1099.977,143.509,-63.651,177.246,15.736,151.903
C04165=1099.971,143.260,-63.631,177.243,15.736,151.903
C04166=1099.966,143.010,-63.610,177.240,15.736,151.904
C04167=1099.960,142.762,-63.590,177.236,15.736,151.905
C04168=1099.954,142.512,-63.569,177.233,15.737,151.906
C04169=1099.949,142.263,-63.549,177.230,15.736,151.906
C04170=1099.944,142.014,-63.528,177.227,15.737,151.907
C04171=1099.938,141.765,-63.508,177.224,15.737,151.908
C04172=1099.932,141.515,-63.487,177.220,15.737,151.908
C04173=1099.927,141.266,-63.467,177.218,15.737,151.909
C04174=1099.921,141.018,-63.447,177.214,15.737,151.910
C04175=1099.915,140.769,-63.425,177.211,15.737,151.910
C04176=1099.909,140.520,-63.405,177.208,15.737,151.911
C04177=1099.904,140.271,-63.385,177.204,15.737,151.912
C04178=1099.899,140.022,-63.364,177.202,15.738,151.912
C04179=1099.892,139.772,-63.345,177.198,15.738,151.913
C04180=1099.887,139.523,-63.324,177.194,15.738,151.914
C04181=1099.881,139.274,-63.304,177.192,15.738,151.914
C04182=1099.876,139.025,-63.284,177.188,15.738,151.915
C04183=1099.870,138.776,-63.264,177.186,15.738,151.916
C04184=1099.865,138.527,-63.243,177.182,15.738,151.917
C04185=1099.859,138.278,-63.223,177.179,15.738,151.917
C04186=1099.853,138.028,-63.202,177.176,15.738,151.918
C04187=1099.847,137.779,-63.182,177.172,15.738,151.919
C04188=1099.841,137.530,-63.162,177.170,15.739,151.919
C04189=1099.835,137.281,-63.142,177.166,15.739,151.920
C04190=1099.830,137.032,-63.121,177.163,15.739,151.921
C04191=1099.825,136.783,-63.102,177.160,15.739,151.921
C04192=1099.819,136.534,-63.081,177.157,15.739,151.922
C04193=1099.813,136.285,-63.061,177.154,15.739,151.923
C04194=1099.808,136.036,-63.041,177.151,15.739,151.923
C04195=1099.802,135.787,-63.021,177.147,15.739,151.924
C04196=1099.796,135.537,-63.000,177.145,15.739,151.925
C04197=1099.790,135.288,-62.981,177.141,15.739,151.925
C04198=1099.785,135.039,-62.960,177.138,15.740,151.926
C04199=1099.779,134.790,-62.940,177.135,15.739,151.927
C04200=1099.773,134.541,-62.920,177.131,15.739,151.927
C04201=1099.768,134.291,-62.900,177.129,15.739,151.928
C04202=1099.762,134.042,-62.880,177.125,15.739,151.929
C04203=1099.757,133.793,-62.860,177.123,15.739,151.929
C04204=1099.751,133.545,-62.840,177.119,15.739,151.930
C04205=1099.746,133.295,-62.820,177.116,15.739,151.931
C04206=1099.740,133.046,-62.800,177.113,15.739,151.931
C04207=1099.734,132.797,-62.780,177.110,15.739,151.932
C04208=1099.729,132.547,-62.760,177.107,15.740,151.933
C04209=1099.723,132.299,-62.740,177.104,15.740,151.933
C04210=1099.717,132.050,-62.720,177.100,15.739,151.934
C04211=1099.712,131.800,-62.701,177.098,15.740,151.935
C04212=1099.706,131.551,-62.681,177.094,15.739,151.935
C04213=1099.700,131.302,-62.661,177.092,15.740,151.936
C04214=1099.695,131.053,-62.641,177.088,15.739,151.937
C04215=1099.689,130.804,-62.621,177.085,15.739,151.937
C04216=1099.683,130.555,-62.601,177.082,15.740,151.938
C04217=1099.678,130.306,-62.582,177.079,15.740,151.939
C04218=1099.672,130.057,-62.562,177.076,15.740,151.939
C04219=1099.666,129.807,-62.542,177.073,15.740,151.940
C04220=1099.661,129.558,-62.522,177.070,15.740,151.940
C04221=1099.655,129.309,-62.502,177.067,15.740,151.941
C04222=1099.649,129.060,-62.483,177.063,15.739,151.942
C04223=1099.643,128.811,-62.463,177.061,15.740,151.943
C04224=1099.637,128.562,-62.444,177.057,15.740,151.943
C04225=1099.631,128.288,-62.421,177.054,15.740,151.944
C04226=1099.625,128.013,-62.400,177.051,15.740,151.945
C04227=1099.618,127.740,-62.378,177.047,15.740,151.945
C04228=1099.612,127.466,-62.356,177.044,15.740,151.946
C04229=1099.606,127.217,-62.337,177.040,15.740,151.947
C04230=1099.600,126.967,-62.318,177.038,15.740,151.947
C04231=1099.595,126.718,-62.297,177.034,15.740,151.948
C04232=1099.589,126.469,-62.278,177.032,15.740,151.949
C04233=1099.583,126.220,-62.258,177.029,15.740,151.949
C04234=1099.578,125.971,-62.239,177.025,15.740,151.950
C04235=1099.572,125.723,-62.219,177.023,15.740,151.950
C04236=1099.567,125.473,-62.200,177.019,15.739,151.951
C04237=1099.561,125.224,-62.181,177.017,15.740,151.952
C04238=1099.555,124.975,-62.161,177.013,15.740,151.952
C04239=1099.550,124.725,-62.141,177.011,15.740,151.953
C04240=1099.544,124.476,-62.121,177.007,15.740,151.954
C04241=1099.538,124.227,-62.102,177.004,15.739,151.954
C04242=1099.533,123.977,-62.082,177.002,15.739,151.955
C04243=1099.527,123.729,-62.062,176.998,15.739,151.956
C04244=1099.521,123.479,-62.043,176.995,15.740,151.956
C04245=1099.516,123.230,-62.024,176.992,15.739,151.957
C04246=1099.510,122.982,-62.004,176.990,15.739,151.957
C04247=1099.504,122.732,-61.985,176.986,15.739,151.958
C04248=1099.499,122.483,-61.966,176.983,15.739,151.959
C04249=1099.493,122.233,-61.947,176.980,15.739,151.959
C04250=1099.487,121.985,-61.927,176.977,15.739,151.960
C04251=1099.482,121.735,-61.907,176.975,15.739,151.960
C04252=1099.477,121.486,-61.888,176.971,15.739,151.961
C04253=1099.471,121.237,-61.869,176.969,15.739,151.962
C04254=1099.465,120.988,-61.849,176.965,15.738,151.962
C04255=1099.460,120.738,-61.829,176.962,15.738,151.963
C04256=1099.454,120.489,-61.810,176.960,15.738,151.963
C04257=1099.449,120.240,-61.791,176.956,15.738,151.964
C04258=1099.443,119.991,-61.772,176.954,15.738,151.965
C04259=1099.437,119.741,-61.753,176.950,15.738,151.965
C04260=1099.431,119.493,-61.733,176.948,15.738,151.966
C04261=1099.426,119.243,-61.714,176.944,15.738,151.966
C04262=1099.421,118.994,-61.695,176.941,15.737,151.967
C04263=1099.415,118.745,-61.676,176.939,15.737,151.967
C04264=1099.409,118.496,-61.656,176.935,15.737,151.968
C04265=1099.404,118.246,-61.637,176.933,15.737,151.969
C04266=1099.398,117.997,-61.618,176.930,15.737,151.969
C04267=1099.393,117.748,-61.599,176.927,15.737,151.970
C04268=1099.387,117.499,-61.579,176.924,15.736,151.970
C04269=1099.381,117.250,-61.560,176.921,15.736,151.971
C04270=1099.376,117.001,-61.541,176.918,15.736,151.971
C04271=1099.370,116.752,-61.522,176.915,15.736,151.972
C04272=1099.365,116.502,-61.502,176.912,15.736,151.973
C04273=1099.359,116.253,-61.483,176.909,15.736,151.973
C04274=1099.353,116.004,-61.465,176.907,15.735,151.974
C04275=1099.347,115.755,-61.446,176.903,15.735,151.974
C04276=1099.342,115.505,-61.426,176.901,15.735,151.975
C04277=1099.337,115.257,-61.407,176.898,15.735,151.976
C04278=1099.331,115.007,-61.388,176.894,15.734,151.976
C04279=1099.325,114.758,-61.369,176.892,15.734,151.977
C04280=1099.320,114.509,-61.350,176.889,15.734,151.977
C04281=1099.314,114.260,-61.331,176.886,15.734,151.978
C04282=1099.309,114.010,-61.312,176.883,15.734,151.978
C04283=1099.303,113.760,-61.294,176.880,15.734,151.979
C04284=1099.298,113.512,-61.275,176.877,15.734,151.980
C04285=1099.292,113.262,-61.256,176.875,15.734,151.980
C04286=1099.286,113.013,-61.236,176.871,15.733,151.981
C04287=1099.281,112.763,-61.217,176.868,15.733,151.981
C04288=1099.275,112.515,-61.199,176.866,15.733,151.982
C04289=1099.269,112.241,-61.178,176.862,15.733,151.982
C04290=1099.262,111.967,-61.157,176.859,15.733,151.983
C04291=1099.256,111.693,-61.136,176.856,15.732,151.984
C04292=1099.250,111.420,-61.115,176.853,15.732,151.984
C04293=1099.244,111.170,-61.097,176.850,15.732,151.985
C04294=1099.239,110.920,-61.078,176.847,15.732,151.986
C04295=1099.233,110.672,-61.059,176.844,15.732,151.986
C04296=1099.227,110.422,-61.040,176.842,15.732,151.987
C04297=1099.222,110.173,-61.021,176.838,15.731,151.987
C04298=1099.216,109.925,-61.003,176.835,15.731,151.988
C04299=1099.210,109.674,-60.984,176.833,15.731,151.988
C04300=1099.204,109.425,-60.965,176.830,15.730,151.989
C04301=1099.199,109.177,-60.947,176.827,15.730,151.989
C04302=1099.193,108.927,-60.927,176.824,15.730,151.990
C04303=1099.187,108.677,-60.909,176.821,15.730,151.991
C04304=1099.182,108.429,-60.891,176.818,15.730,151.991
C04305=1099.176,108.179,-60.871,176.816,15.730,151.992
C04306=1099.170,107.930,-60.853,176.812,15.729,151.992
C04307=1099.165,107.681,-60.834,176.810,15.729,151.993
C04308=1099.159,107.432,-60.816,176.807,15.729,151.993
C04309=1099.153,107.182,-60.797,176.804,15.729,151.994
C04310=1099.148,106.933,-60.778,176.801,15.728,151.994
C04311=1099.142,106.684,-60.760,176.799,15.729,151.995
C04312=1099.137,106.435,-60.741,176.796,15.728,151.995
C04313=1099.131,106.185,-60.723,176.792,15.727,151.996
C04314=1099.125,105.936,-60.704,176.790,15.727,151.997
C04315=1099.119,105.687,-60.686,176.787,15.727,151.997
C04316=1099.114,105.437,-60.667,176.784,15.727,151.998
C04317=1099.109,105.189,-60.648,176.781,15.726,151.998
C04318=1099.102,104.939,-60.630,176.779,15.726,151.999
C04319=1099.097,104.690,-60.611,176.775,15.726,151.999
C04320=1099.091,104.440,-60.593,176.773,15.726,152.000
C04321=1099.086,104.191,-60.574,176.770,15.725,152.000
C04322=1099.080,103.943,-60.556,176.768,15.726,152.001
C04323=1099.074,103.693,-60.537,176.764,15.725,152.001
C04324=1099.068,103.444,-60.519,176.762,15.725,152.002
C04325=1099.063,103.194,-60.500,176.759,15.724,152.002
C04326=1099.057,102.946,-60.482,176.756,15.725,152.003
C04327=1099.052,102.696,-60.464,176.753,15.724,152.003
C04328=1099.046,102.447,-60.445,176.751,15.724,152.004
C04329=1099.041,102.197,-60.427,176.748,15.723,152.004
C04330=1099.035,101.949,-60.409,176.745,15.723,152.005
C04331=1099.029,101.699,-60.390,176.742,15.723,152.006
C04332=1099.024,101.450,-60.372,176.739,15.722,152.006
C04333=1099.018,101.200,-60.353,176.737,15.722,152.007
C04334=1099.012,100.950,-60.335,176.733,15.722,152.007
C04335=1099.007,100.702,-60.316,176.731,15.721,152.008
C04336=1099.001,100.452,-60.298,176.728,15.721,152.008
C04337=1098.995,100.204,-60.280,176.725,15.721,152.009
C04338=1098.990,99.954,-60.262,176.722,15.720,152.009
C04339=1098.984,99.705,-60.243,176.720,15.720,152.010
C04340=1098.978,99.455,-60.225,176.717,15.720,152.010
C04341=1098.973,99.206,-60.207,176.715,15.720,152.011
C04342=1098.967,98.957,-60.189,176.711,15.719,152.011
C04343=1098.961,98.708,-60.171,176.709,15.719,152.012
C04344=1098.956,98.458,-60.153,176.706,15.719,152.012
C04345=1098.950,98.209,-60.134,176.703,15.719,152.013
C04346=1098.944,97.960,-60.116,176.700,15.718,152.013
C04347=1098.939,97.710,-60.098,176.698,15.718,152.014
C04348=1098.933,97.461,-60.079,176.695,15.717,152.014
C04349=1098.927,97.212,-60.062,176.692,15.717,152.015
C04350=1098.922,96.962,-60.043,176.689,15.716,152.015
C04351=1098.916,96.714,-60.025,176.687,15.717,152.016
C04352=1098.910,96.464,-60.007,176.684,15.716,152.016
C04353=1098.904,96.190,-59.987,176.681,15.715,152.017
C04354=1098.898,95.917,-59.967,176.678,15.715,152.017
C04355=1098.891,95.643,-59.948,176.675,15.715,152.018
C04356=1098.885,95.369,-59.928,176.672,15.714,152.018
C04357=1098.879,95.119,-59.910,176.670,15.714,152.019
C04358=1098.874,94.871,-59.892,176.667,15.713,152.019
C04359=1098.869,94.621,-59.874,176.664,15.714,152.020
C04360=1098.863,94.372,-59.856,176.661,15.713,152.020
C04361=1098.857,94.123,-59.838,176.659,15.713,152.021
C04362=1098.851,93.873,-59.820,176.656,15.712,152.021
C04363=1098.846,93.623,-59.802,176.653,15.712,152.022
C04364=1098.840,93.375,-59.784,176.650,15.711,152.022
C04365=1098.834,93.125,-59.766,176.648,15.711,152.023
C04366=1098.829,92.876,-59.748,176.645,15.711,152.023
C04367=1098.823,92.626,-59.730,176.643,15.710,152.024
C04368=1098.818,92.377,-59.712,176.639,15.710,152.024
C04369=1098.812,92.128,-59.695,176.637,15.710,152.025
C04370=1098.806,91.878,-59.677,176.634,15.709,152.025
C04371=1098.801,91.629,-59.659,176.632,15.709,152.026
C04372=1098.796,91.380,-59.641,176.629,15.708,152.026
C04373=1098.789,91.131,-59.622,176.627,15.708,152.027
C04374=1098.784,90.882,-59.605,176.623,15.707,152.027
C04375=1098.778,90.632,-59.587,176.621,15.707,152.028
C04376=1098.772,90.383,-59.569,176.618,15.706,152.028
C04377=1098.767,90.134,-59.552,176.616,15.706,152.029
C04378=1098.761,89.884,-59.534,176.613,15.706,152.029
C04379=1098.755,89.635,-59.516,176.610,15.706,152.030
C04380=1098.750,89.386,-59.498,176.607,15.705,152.030
C04381=1098.744,89.136,-59.481,176.605,15.705,152.031
C04382=1098.738,88.887,-59.463,176.602,15.704,152.031
C04383=1098.732,88.638,-59.445,176.600,15.704,152.032
C04384=1098.726,88.389,-59.427,176.597,15.703,152.032
C04385=1098.721,88.140,-59.410,176.594,15.703,152.033
C04386=1098.715,87.890,-59.392,176.591,15.702,152.033
C04387=1098.709,87.641,-59.374,176.589,15.702,152.033
C04388=1098.704,87.392,-59.357,176.586,15.702,152.034
C04389=1098.698,87.142,-59.339,176.583,15.701,152.034
C04390=1098.692,86.892,-59.322,176.581,15.701,152.035
C04391=1098.687,86.643,-59.305,176.578,15.701,152.035
C04392=1098.681,86.394,-59.287,176.575,15.700,152.036
C04393=1098.675,86.145,-59.269,176.573,15.700,152.036
C04394=1098.670,85.895,-59.251,176.571,15.699,152.037
C04395=1098.664,85.646,-59.234,176.567,15.699,152.037
C04396=1098.658,85.397,-59.216,176.565,15.699,152.038
C04397=1098.653,85.148,-59.198,176.562,15.698,152.038
C04398=1098.647,84.899,-59.181,176.560,15.697,152.038
C04399=1098.641,84.648,-59.164,176.557,15.697,152.039
C04400=1098.636,84.399,-59.146,176.555,15.697,152.039
C04401=1098.630,84.150,-59.128,176.552,15.696,152.040
C04402=1098.625,83.901,-59.111,176.549,15.696,152.040
C04403=1098.619,83.651,-59.093,176.546,15.695,152.041
C04404=1098.613,83.402,-59.076,176.544,15.695,152.041
C04405=1098.608,83.153,-59.059,176.541,15.694,152.042
C04406=1098.602,82.904,-59.041,176.539,15.694,152.042
C04407=1098.595,82.654,-59.024,176.536,15.693,152.043
C04408=1098.590,82.405,-59.007,176.534,15.693,152.043
C04409=1098.585,82.156,-58.989,176.531,15.692,152.043
C04410=1098.579,81.906,-58.972,176.529,15.692,152.044
C04411=1098.574,81.657,-58.954,176.526,15.691,152.044
C04412=1098.568,81.407,-58.937,176.523,15.691,152.045
C04413=1098.562,81.158,-58.919,176.521,15.691,152.045
C04414=1098.557,80.909,-58.902,176.518,15.690,152.046
C04415=1098.552,80.659,-58.885,176.516,15.689,152.046
C04416=1098.546,80.410,-58.867,176.513,15.689,152.046
C04417=1098.539,80.136,-58.848,176.510,15.688,152.047
C04418=1098.533,79.863,-58.829,176.508,15.687,152.047
C04419=1098.527,79.589,-58.811,176.504,15.687,152.048
C04420=1098.520,79.315,-58.791,176.501,15.686,152.048
C04421=1098.515,79.066,-58.774,176.499,15.686,152.049
C04422=1098.510,78.816,-58.757,176.496,15.685,152.049
C04423=1098.504,78.567,-58.739,176.494,15.685,152.050
C04424=1098.499,78.318,-58.722,176.491,15.684,152.050
C04425=1098.493,78.069,-58.705,176.489,15.684,152.050
C04426=1098.486,77.819,-58.688,176.487,15.683,152.051
C04427=1098.481,77.569,-58.671,176.484,15.682,152.051
C04428=1098.476,77.320,-58.653,176.482,15.682,152.052
C04429=1098.470,77.071,-58.637,176.479,15.681,152.052
C04430=1098.464,76.822,-58.619,176.476,15.681,152.053
C04431=1098.458,76.572,-58.602,176.473,15.681,152.053
C04432=1098.452,76.323,-58.585,176.471,15.680,152.054
C04433=1098.447,76.073,-58.568,176.468,15.680,152.054
C04434=1098.441,75.824,-58.551,176.466,15.679,152.054
C04435=1098.435,75.575,-58.534,176.463,15.678,152.055
C04436=1098.430,75.326,-58.517,176.461,15.678,152.055
C04437=1098.425,75.076,-58.500,176.458,15.678,152.056
C04438=1098.418,74.827,-58.483,176.455,15.677,152.056
C04439=1098.413,74.577,-58.466,176.453,15.677,152.056
C04440=1098.407,74.328,-58.448,176.450,15.676,152.057
C04441=1098.401,74.079,-58.432,176.448,15.675,152.057
C04442=1098.396,73.830,-58.414,176.445,15.674,152.058
C04443=1098.390,73.580,-58.398,176.443,15.674,152.058
C04444=1098.384,73.331,-58.381,176.440,15.673,152.058
C04445=1098.379,73.082,-58.364,176.438,15.673,152.059
C04446=1098.373,72.831,-58.347,176.436,15.673,152.059
C04447=1098.367,72.582,-58.330,176.433,15.672,152.060
C04448=1098.362,72.333,-58.313,176.431,15.671,152.060
C04449=1098.355,72.084,-58.296,176.428,15.671,152.061
C04450=1098.350,71.834,-58.279,176.426,15.670,152.061
C04451=1098.345,71.585,-58.262,176.423,15.669,152.061
C04452=1098.339,71.336,-58.245,176.420,15.669,152.062
C04453=1098.334,71.086,-58.228,176.418,15.668,152.062
C04454=1098.328,70.837,-58.212,176.416,15.668,152.062
C04455=1098.322,70.588,-58.194,176.413,15.667,152.063
C04456=1098.317,70.338,-58.178,176.410,15.666,152.063
C04457=1098.311,70.089,-58.161,176.408,15.666,152.064
C04458=1098.305,69.840,-58.144,176.405,15.665,152.064
C04459=1098.299,69.591,-58.127,176.403,15.665,152.065
C04460=1098.294,69.341,-58.111,176.400,15.664,152.065
C04461=1098.288,69.091,-58.094,176.398,15.663,152.065
C04462=1098.282,68.842,-58.076,176.396,15.663,152.066
C04463=1098.276,68.592,-58.060,176.393,15.662,152.066
C04464=1098.271,68.343,-58.043,176.391,15.662,152.067
C04465=1098.265,68.093,-58.027,176.388,15.661,152.067
C04466=1098.260,67.844,-58.010,176.386,15.660,152.067
C04467=1098.254,67.595,-57.993,176.383,15.660,152.068
C04468=1098.248,67.345,-57.976,176.381,15.659,152.068
C04469=1098.242,67.096,-57.960,176.378,15.658,152.069
C04470=1098.236,66.847,-57.943,176.376,15.658,152.069
C04471=1098.231,66.598,-57.926,176.374,15.658,152.069
C04472=1098.225,66.348,-57.910,176.371,15.657,152.070
C04473=1098.220,66.099,-57.893,176.369,15.656,152.070
C04474=1098.214,65.849,-57.877,176.366,15.655,152.070
C04475=1098.209,65.600,-57.860,176.364,15.655,152.071
C04476=1098.202,65.351,-57.843,176.362,15.654,152.071
C04477=1098.196,65.102,-57.827,176.359,15.654,152.072
C04478=1098.191,64.852,-57.810,176.357,15.653,152.072
C04479=1098.185,64.603,-57.794,176.354,15.652,152.072
C04480=1098.179,64.353,-57.778,176.352,15.652,152.073
C04481=1098.174,64.079,-57.759,176.349,15.651,152.073
C04482=1098.167,63.805,-57.741,176.347,15.651,152.073
C04483=1098.161,63.531,-57.723,176.344,15.650,152.074
C04484=1098.155,63.258,-57.705,176.341,15.649,152.074
C04485=1098.149,63.008,-57.689,176.338,15.649,152.075
C04486=1098.143,62.760,-57.672,176.335,15.648,152.075
C04487=1098.137,62.510,-57.655,176.333,15.648,152.076
C04488=1098.131,62.261,-57.639,176.331,15.647,152.076
C04489=1098.126,62.011,-57.622,176.328,15.646,152.076
C04490=1098.120,61.762,-57.606,176.326,15.646,152.077
C04491=1098.114,61.513,-57.590,176.323,15.645,152.077
C04492=1098.108,61.263,-57.574,176.321,15.644,152.077
C04493=1098.102,61.014,-57.557,176.319,15.644,152.078
C04494=1098.097,60.764,-57.540,176.316,15.643,152.078
C04495=1098.091,60.515,-57.524,176.314,15.643,152.079
C04496=1098.085,60.266,-57.508,176.311,15.641,152.079
C04497=1098.079,60.016,-57.492,176.309,15.641,152.079
C04498=1098.073,59.767,-57.475,176.307,15.641,152.080
C04499=1098.067,59.517,-57.459,176.304,15.640,152.080
C04500=1098.062,59.267,-57.443,176.302,15.639,152.080
C04501=1098.056,59.018,-57.427,176.299,15.638,152.081
C04502=1098.050,58.768,-57.411,176.297,15.638,152.081
C04503=1098.044,58.519,-57.394,176.295,15.637,152.082
C04504=1098.039,58.269,-57.377,176.292,15.637,152.082
C04505=1098.033,58.020,-57.361,176.290,15.636,152.082
C04506=1098.027,57.771,-57.345,176.287,15.635,152.083
C04507=1098.021,57.521,-57.329,176.285,15.634,152.083
C04508=1098.016,57.273,-57.313,176.283,15.634,152.083
C04509=1098.010,57.023,-57.297,176.280,15.633,152.084
C04510=1098.005,56.773,-57.280,176.278,15.632,152.084
C04511=1097.999,56.524,-57.264,176.275,15.632,152.084
C04512=1097.993,56.274,-57.248,176.273,15.631,152.085
C04513=1097.987,56.025,-57.232,176.271,15.631,152.085
C04514=1097.981,55.776,-57.215,176.268,15.630,152.086
C04515=1097.975,55.526,-57.200,176.266,15.629,152.086
C04516=1097.970,55.277,-57.184,176.263,15.628,152.086
C04517=1097.964,55.028,-57.168,176.262,15.627,152.087
C04518=1097.959,54.778,-57.151,176.259,15.627,152.087
C04519=1097.953,54.529,-57.135,176.257,15.626,152.087
C04520=1097.947,54.279,-57.119,176.255,15.626,152.088
C04521=1097.941,54.029,-57.103,176.253,15.625,152.088
C04522=1097.936,53.781,-57.087,176.250,15.624,152.088
C04523=1097.930,53.531,-57.071,176.248,15.623,152.089
C04524=1097.924,53.282,-57.055,176.245,15.622,152.089
C04525=1097.918,53.032,-57.039,176.243,15.622,152.089
C04526=1097.912,52.783,-57.023,176.241,15.621,152.090
C04527=1097.907,52.533,-57.007,176.238,15.620,152.090
C04528=1097.901,52.284,-56.991,176.236,15.620,152.090
C04529=1097.895,52.035,-56.975,176.233,15.618,152.091
C04530=1097.891,51.785,-56.959,176.231,15.618,152.091
C04531=1097.885,51.535,-56.942,176.229,15.617,152.091
C04532=1097.879,51.286,-56.926,176.226,15.617,152.092
C04533=1097.874,51.037,-56.911,176.224,15.616,152.092
C04534=1097.868,50.787,-56.895,176.222,15.616,152.092
C04535=1097.862,50.538,-56.879,176.219,15.614,152.093
C04536=1097.856,50.288,-56.863,176.217,15.614,152.093
C04537=1097.851,50.039,-56.847,176.215,15.613,152.093
C04538=1097.845,49.790,-56.831,176.213,15.612,152.094
C04539=1097.839,49.540,-56.815,176.211,15.612,152.094
C04540=1097.833,49.291,-56.799,176.208,15.610,152.094
C04541=1097.828,49.041,-56.784,176.206,15.610,152.095
C04542=1097.822,48.792,-56.768,176.204,15.609,152.095
C04543=1097.816,48.542,-56.752,176.201,15.608,152.095
C04544=1097.811,48.293,-56.736,176.199,15.608,152.096
C04545=1097.804,48.019,-56.719,176.196,15.607,152.096
C04546=1097.799,47.745,-56.701,176.194,15.606,152.096
C04547=1097.792,47.471,-56.684,176.191,15.605,152.097
C04548=1097.786,47.197,-56.667,176.188,15.604,152.097
C04549=1097.780,46.947,-56.651,176.187,15.603,152.097
C04550=1097.775,46.697,-56.635,176.185,15.603,152.098
C04551=1097.769,46.449,-56.619,176.182,15.602,152.098
C04552=1097.764,46.199,-56.604,176.180,15.601,152.098
C04553=1097.758,45.949,-56.587,176.178,15.600,152.099
C04554=1097.753,45.700,-56.572,176.175,15.600,152.099
C04555=1097.747,45.451,-56.556,176.173,15.599,152.099
C04556=1097.741,45.201,-56.541,176.170,15.597,152.100
C04557=1097.736,44.952,-56.525,176.169,15.597,152.100
C04558=1097.730,44.702,-56.509,176.166,15.596,152.100
C04559=1097.724,44.452,-56.494,176.164,15.595,152.100
C04560=1097.719,44.204,-56.478,176.162,15.594,152.101
C04561=1097.713,43.954,-56.462,176.160,15.594,152.101
C04562=1097.708,43.705,-56.446,176.157,15.593,152.101
C04563=1097.702,43.455,-56.431,176.155,15.592,152.102
C04564=1097.696,43.205,-56.416,176.153,15.591,152.102
C04565=1097.690,42.956,-56.399,176.150,15.591,152.102
C04566=1097.685,42.707,-56.384,176.148,15.590,152.103
C04567=1097.679,42.457,-56.369,176.146,15.588,152.103
C04568=1097.673,42.208,-56.353,176.143,15.588,152.103
C04569=1097.668,41.958,-56.338,176.142,15.588,152.104
C04570=1097.662,41.708,-56.322,176.139,15.586,152.104
C04571=1097.656,41.459,-56.306,176.137,15.586,152.104
C04572=1097.650,41.210,-56.292,176.135,15.585,152.104
C04573=1097.645,40.960,-56.276,176.132,15.584,152.105
C04574=1097.639,40.712,-56.260,176.130,15.583,152.105
C04575=1097.634,40.462,-56.245,176.128,15.583,152.105
C04576=1097.627,40.212,-56.230,176.125,15.582,152.106
C04577=1097.622,39.963,-56.214,176.124,15.581,152.106
C04578=1097.616,39.713,-56.198,176.122,15.580,152.106
C04579=1097.611,39.463,-56.183,176.119,15.579,152.107
C04580=1097.605,39.214,-56.168,176.117,15.579,152.107
C04581=1097.599,38.965,-56.152,176.115,15.578,152.107
C04582=1097.594,38.716,-56.137,176.112,15.577,152.107
C04583=1097.588,38.466,-56.121,176.110,15.576,152.108
C04584=1097.582,38.216,-56.106,176.108,15.576,152.108
C04585=1097.577,37.967,-56.091,176.106,15.574,152.108
C04586=1097.571,37.717,-56.075,176.104,15.574,152.109
C04587=1097.565,37.469,-56.060,176.102,15.573,152.109
C04588=1097.559,37.219,-56.045,176.099,15.572,152.109
C04589=1097.553,36.969,-56.030,176.097,15.571,152.110
C04590=1097.548,36.720,-56.014,176.095,15.570,152.110
C04591=1097.542,36.470,-55.998,176.092,15.569,152.110
C04592=1097.536,36.221,-55.983,176.090,15.569,152.111
C04593=1097.530,35.971,-55.968,176.088,15.568,152.111
C04594=1097.524,35.722,-55.953,176.086,15.567,152.111
C04595=1097.519,35.472,-55.938,176.084,15.566,152.111
C04596=1097.513,35.223,-55.923,176.082,15.565,152.112
C04597=1097.508,34.974,-55.908,176.079,15.565,152.112
C04598=1097.502,34.724,-55.892,176.077,15.564,152.112
C04599=1097.495,34.475,-55.877,176.075,15.563,152.113
C04600=1097.490,34.225,-55.862,176.072,15.562,152.113
C04601=1097.484,33.976,-55.847,176.071,15.561,152.113
C04602=1097.479,33.726,-55.831,176.068,15.561,152.113
C04603=1097.472,33.477,-55.816,176.066,15.560,152.114
C04604=1097.467,33.227,-55.801,176.064,15.559,152.114
C04605=1097.461,32.978,-55.786,176.062,15.558,152.114
C04606=1097.455,32.728,-55.771,176.060,15.557,152.115
C04607=1097.450,32.479,-55.756,176.057,15.556,152.115
C04608=1097.444,32.229,-55.741,176.055,15.555,152.115
C04609=1097.438,31.955,-55.724,176.052,15.554,152.116
C04610=1097.432,31.681,-55.707,176.051,15.554,152.116
C04611=1097.425,31.408,-55.691,176.048,15.552,152.116
C04612=1097.419,31.133,-55.675,176.046,15.552,152.116
C04613=1097.413,30.883,-55.660,176.043,15.550,152.117
C04614=1097.408,30.634,-55.645,176.041,15.550,152.117
C04615=1097.401,30.384,-55.630,176.039,15.549,152.117
C04616=1097.396,30.135,-55.615,176.037,15.548,152.118
C04617=1097.390,29.885,-55.600,176.035,15.547,152.118
C04618=1097.385,29.636,-55.584,176.033,15.547,152.118
C04619=1097.379,29.386,-55.569,176.031,15.546,152.118
C04620=1097.374,29.137,-55.554,176.028,15.545,152.119
C04621=1097.367,28.888,-55.539,176.026,15.544,152.119
C04622=1097.362,28.638,-55.524,176.025,15.543,152.119
C04623=1097.356,28.389,-55.509,176.022,15.542,152.119
C04624=1097.351,28.139,-55.494,176.020,15.541,152.120
C04625=1097.345,27.889,-55.480,176.018,15.540,152.120
C04626=1097.339,27.640,-55.465,176.015,15.540,152.120
C04627=1097.333,27.390,-55.450,176.013,15.539,152.121
C04628=1097.327,27.141,-55.435,176.011,15.538,152.121
C04629=1097.321,26.892,-55.420,176.009,15.537,152.121
C04630=1097.316,26.642,-55.405,176.007,15.536,152.121
C04631=1097.310,26.393,-55.390,176.005,15.535,152.122
C04632=1097.304,26.143,-55.376,176.003,15.535,152.122
C04633=1097.299,25.894,-55.361,176.000,15.533,152.122
C04634=1097.293,25.644,-55.346,175.999,15.533,152.122
C04635=1097.287,25.395,-55.331,175.997,15.532,152.123
C04636=1097.281,25.145,-55.316,175.995,15.531,152.123
C04637=1097.276,24.896,-55.302,175.992,15.530,152.123
C04638=1097.269,24.646,-55.287,175.990,15.529,152.123
C04639=1097.264,24.397,-55.272,175.988,15.528,152.124
C04640=1097.258,24.147,-55.257,175.986,15.527,152.124
C04641=1097.253,23.897,-55.243,175.984,15.526,152.124
C04642=1097.247,23.648,-55.229,175.982,15.526,152.125
C04643=1097.241,23.399,-55.213,175.980,15.525,152.125
C04644=1097.235,23.150,-55.198,175.977,15.524,152.125
C04645=1097.229,22.899,-55.184,175.975,15.523,152.125
C04646=1097.224,22.650,-55.169,175.974,15.522,152.126
C04647=1097.218,22.401,-55.154,175.971,15.521,152.126
C04648=1097.212,22.151,-55.140,175.969,15.520,152.126
C04649=1097.207,21.902,-55.126,175.967,15.519,152.126
C04650=1097.201,21.652,-55.110,175.965,15.519,152.127
C04651=1097.195,21.403,-55.096,175.963,15.517,152.127
C04652=1097.190,21.153,-55.082,175.961,15.517,152.127
C04653=1097.183,20.904,-55.067,175.959,15.516,152.127
C04654=1097.178,20.654,-55.052,175.957,15.515,152.128
C04655=1097.172,20.404,-55.037,175.954,15.514,152.128
C04656=1097.166,20.155,-55.023,175.952,15.513,152.128
C04657=1097.161,19.906,-55.009,175.950,15.512,152.128
C04658=1097.155,19.656,-54.994,175.948,15.511,152.129
C04659=1097.149,19.407,-54.979,175.946,15.510,152.129
C04660=1097.144,19.157,-54.965,175.944,15.510,152.129
C04661=1097.138,18.907,-54.950,175.942,15.509,152.130
C04662=1097.132,18.658,-54.936,175.939,15.508,152.130
C04663=1097.126,18.408,-54.921,175.938,15.507,152.130
C04664=1097.120,18.159,-54.907,175.936,15.506,152.130
C04665=1097.115,17.910,-54.893,175.934,15.505,152.131
C04666=1097.108,17.660,-54.878,175.931,15.504,152.131
C04667=1097.103,17.410,-54.863,175.929,15.503,152.131
C04668=1097.098,17.161,-54.849,175.927,15.503,152.131
C04669=1097.092,16.911,-54.834,175.925,15.502,152.132
C04670=1097.086,16.662,-54.820,175.923,15.500,152.132
C04671=1097.080,16.412,-54.806,175.921,15.499,152.132
C04672=1097.074,16.163,-54.791,175.919,15.499,152.132
C04673=1097.068,15.890,-54.776,175.917,15.497,152.133
C04674=1097.062,15.617,-54.760,175.915,15.497,152.133
C04675=1097.056,15.345,-54.744,175.912,15.495,152.133
C04676=1097.049,15.072,-54.729,175.910,15.495,152.133
C04677=1097.043,14.823,-54.714,175.908,15.494,152.134
C04678=1097.038,14.573,-54.699,175.906,15.493,152.134
C04679=1097.032,14.324,-54.685,175.904,15.492,152.134
C04680=1097.027,14.074,-54.671,175.902,15.491,152.134
C04681=1097.019,13.825,-54.657,175.900,15.491,152.135
C04682=1097.014,13.575,-54.643,175.898,15.490,152.135
C04683=1097.008,13.326,-54.629,175.895,15.488,152.135
C04684=1097.002,13.076,-54.614,175.894,15.488,152.135
C04685=1096.997,12.826,-54.600,175.892,15.487,152.136
C04686=1096.991,12.577,-54.585,175.890,15.486,152.136
C04687=1096.985,12.327,-54.571,175.887,15.485,152.136
C04688=1096.979,12.078,-54.557,175.886,15.484,152.136
C04689=1096.974,11.829,-54.543,175.884,15.483,152.137
C04690=1096.968,11.579,-54.529,175.882,15.482,152.137
C04691=1096.962,11.329,-54.514,175.879,15.481,152.137
C04692=1096.956,11.080,-54.500,175.877,15.480,152.137
C04693=1096.951,10.830,-54.486,175.875,15.480,152.138
C04694=1096.944,10.581,-54.472,175.873,15.479,152.138
C04695=1096.938,10.331,-54.458,175.871,15.478,152.138
C04696=1096.933,10.082,-54.444,175.869,15.477,152.138
C04697=1096.926,9.832,-54.429,175.867,15.476,152.139
C04698=1096.921,9.582,-54.415,175.865,15.475,152.139
C04699=1096.915,9.333,-54.401,175.864,15.474,152.139
C04700=1096.910,9.083,-54.388,175.861,15.473,152.139
C04701=1096.903,8.834,-54.373,175.859,15.472,152.140
C04702=1096.897,8.584,-54.359,175.857,15.472,152.140
C04703=1096.892,8.335,-54.345,175.855,15.471,152.140
C04704=1096.886,8.086,-54.331,175.853,15.469,152.140
C04705=1096.880,7.836,-54.317,175.851,15.468,152.141
C04706=1096.874,7.586,-54.303,175.849,15.468,152.141
C04707=1096.869,7.336,-54.289,175.847,15.467,152.141
C04708=1096.863,7.088,-54.274,175.845,15.466,152.141
C04709=1096.857,6.838,-54.261,175.843,15.465,152.142
C04710=1096.851,6.588,-54.247,175.841,15.464,152.142
C04711=1096.845,6.338,-54.233,175.839,15.463,152.142
C04712=1096.840,6.089,-54.219,175.837,15.462,152.142
C04713=1096.834,5.840,-54.205,175.835,15.461,152.142
C04714=1096.829,5.590,-54.191,175.833,15.460,152.143
C04715=1096.822,5.340,-54.177,175.831,15.459,152.143
C04716=1096.816,5.091,-54.163,175.829,15.458,152.143
C04717=1096.811,4.841,-54.149,175.827,15.458,152.143
C04718=1096.805,4.592,-54.135,175.825,15.456,152.144
C04719=1096.800,4.342,-54.122,175.823,15.455,152.144
C04720=1096.793,4.093,-54.107,175.821,15.455,152.144
C04721=1096.787,3.843,-54.093,175.819,15.454,152.144
C04722=1096.782,3.594,-54.080,175.818,15.453,152.144
C04723=1096.776,3.344,-54.066,175.815,15.452,152.145
C04724=1096.771,3.094,-54.052,175.813,15.451,152.145
C04725=1096.765,2.845,-54.039,175.811,15.450,152.145
C04726=1096.759,2.596,-54.025,175.810,15.449,152.145
C04727=1096.753,2.345,-54.010,175.808,15.448,152.146
C04728=1096.748,2.096,-53.997,175.805,15.447,152.146
C04729=1096.742,1.846,-53.983,175.803,15.446,152.146
C04730=1096.736,1.597,-53.969,175.802,15.445,152.146
C04731=1096.730,1.348,-53.955,175.800,15.444,152.147
C04732=1096.725,1.098,-53.941,175.798,15.444,152.147
C04733=1096.719,0.849,-53.927,175.795,15.442,152.147
C04734=1096.713,0.599,-53.914,175.793,15.441,152.147
C04735=1096.707,0.349,-53.900,175.792,15.440,152.147
C04736=1096.701,0.100,-53.886,175.790,15.440,152.148
C04737=1096.696,-0.171,-53.872,175.787,15.438,152.148
C04738=1096.689,-0.441,-53.857,175.785,15.437,152.148
C04739=1096.683,-0.712,-53.841,175.784,15.436,152.148
C04740=1096.677,-0.983,-53.826,175.781,15.435,152.149
C04741=1096.671,-1.232,-53.812,175.779,15.434,152.149
C04742=1096.665,-1.482,-53.800,175.777,15.433,152.149
C04743=1096.660,-1.732,-53.786,175.776,15.432,152.149
C04744=1096.655,-1.981,-53.772,175.773,15.431,152.150
C04745=1096.648,-2.231,-53.759,175.771,15.430,152.150
C04746=1096.643,-2.480,-53.745,175.769,15.429,152.150
C04747=1096.637,-2.730,-53.731,175.768,15.429,152.150
C04748=1096.632,-2.979,-53.717,175.766,15.427,152.150
C04749=1096.626,-3.229,-53.704,175.764,15.427,152.150
C04750=1096.620,-3.478,-53.690,175.761,15.425,152.151
C04751=1096.613,-3.728,-53.676,175.760,15.424,152.151
C04752=1096.608,-3.978,-53.663,175.758,15.423,152.151
C04753=1096.602,-4.227,-53.649,175.756,15.423,152.151
C04754=1096.597,-4.477,-53.636,175.754,15.422,152.152
C04755=1096.590,-4.726,-53.623,175.752,15.421,152.152
C04756=1096.585,-4.976,-53.609,175.750,15.419,152.152
C04757=1096.579,-5.225,-53.596,175.748,15.419,152.152
C04758=1096.573,-5.475,-53.582,175.746,15.418,152.153
C04759=1096.567,-5.724,-53.569,175.744,15.417,152.153
C04760=1096.561,-5.974,-53.555,175.743,15.416,152.153
C04761=1096.555,-6.224,-53.542,175.741,15.415,152.153
C04762=1096.549,-6.474,-53.528,175.738,15.414,152.153
C04763=1096.543,-6.723,-53.515,175.736,15.413,152.154
C04764=1096.538,-6.973,-53.501,175.735,15.412,152.154
C04765=1096.532,-7.222,-53.488,175.733,15.411,152.154
C04766=1096.526,-7.472,-53.474,175.731,15.411,152.154
C04767=1096.520,-7.721,-53.461,175.729,15.410,152.154
C04768=1096.515,-7.971,-53.447,175.727,15.408,152.155
C04769=1096.508,-8.220,-53.434,175.725,15.408,152.155
C04770=1096.503,-8.470,-53.420,175.723,15.407,152.155
C04771=1096.497,-8.720,-53.408,175.721,15.406,152.155
C04772=1096.492,-8.969,-53.394,175.719,15.405,152.156
C04773=1096.485,-9.219,-53.380,175.718,15.404,152.156
C04774=1096.480,-9.468,-53.368,175.715,15.402,152.156
C04775=1096.474,-9.718,-53.354,175.713,15.402,152.156
C04776=1096.468,-9.967,-53.341,175.711,15.401,152.156
C04777=1096.462,-10.217,-53.327,175.710,15.400,152.157
C04778=1096.456,-10.467,-53.314,175.708,15.399,152.157
C04779=1096.451,-10.716,-53.300,175.706,15.398,152.157
C04780=1096.445,-10.966,-53.287,175.704,15.398,152.157
C04781=1096.439,-11.215,-53.275,175.702,15.396,152.157
C04782=1096.433,-11.465,-53.261,175.700,15.395,152.158
C04783=1096.427,-11.714,-53.248,175.698,15.394,152.158
C04784=1096.422,-11.965,-53.234,175.696,15.393,152.158
C04785=1096.416,-12.214,-53.221,175.695,15.393,152.158
C04786=1096.410,-12.463,-53.208,175.693,15.392,152.159
C04787=1096.404,-12.713,-53.195,175.691,15.391,152.159
C04788=1096.398,-12.963,-53.181,175.688,15.389,152.159
C04789=1096.393,-13.213,-53.168,175.687,15.389,152.159
C04790=1096.387,-13.462,-53.155,175.685,15.387,152.159
C04791=1096.381,-13.711,-53.142,175.683,15.387,152.160
C04792=1096.375,-13.961,-53.129,175.681,15.386,152.160
C04793=1096.370,-14.210,-53.116,175.680,15.385,152.160
C04794=1096.365,-14.460,-53.103,175.678,15.384,152.160
C04795=1096.358,-14.709,-53.089,175.675,15.382,152.160
C04796=1096.352,-14.959,-53.076,175.674,15.382,152.161
C04797=1096.347,-15.209,-53.063,175.672,15.381,152.161
C04798=1096.341,-15.458,-53.050,175.670,15.380,152.161
C04799=1096.335,-15.708,-53.037,175.668,15.379,152.161
C04800=1096.329,-15.957,-53.024,175.666,15.378,152.161
C04801=1096.322,-16.227,-53.009,175.664,15.377,152.162
C04802=1096.317,-16.496,-52.995,175.662,15.376,152.162
C04803=1096.310,-16.765,-52.982,175.660,15.375,152.162
C04804=1096.303,-17.034,-52.967,175.658,15.374,152.162
C04805=1096.298,-17.284,-52.954,175.656,15.374,152.163
C04806=1096.291,-17.533,-52.941,175.654,15.372,152.163
C04807=1096.285,-17.783,-52.929,175.652,15.371,152.163
C04808=1096.280,-18.032,-52.915,175.650,15.370,152.163
C04809=1096.275,-18.281,-52.903,175.649,15.369,152.163
C04810=1096.269,-18.531,-52.890,175.647,15.369,152.164
C04811=1096.263,-18.781,-52.877,175.645,15.368,152.164
C04812=1096.257,-19.030,-52.864,175.643,15.367,152.164
C04813=1096.251,-19.280,-52.850,175.641,15.366,152.164
C04814=1096.245,-19.530,-52.838,175.639,15.365,152.165
C04815=1096.239,-19.779,-52.824,175.637,15.363,152.165
C04816=1096.233,-20.029,-52.812,175.635,15.363,152.165
C04817=1096.227,-20.278,-52.799,175.633,15.362,152.165
C04818=1096.221,-20.528,-52.786,175.632,15.361,152.165
C04819=1096.216,-20.778,-52.773,175.630,15.360,152.166
C04820=1096.210,-21.027,-52.760,175.628,15.359,152.166
C04821=1096.204,-21.277,-52.747,175.626,15.358,152.166
C04822=1096.198,-21.526,-52.734,175.625,15.357,152.166
C04823=1096.192,-21.776,-52.722,175.623,15.357,152.166
C04824=1096.186,-22.026,-52.709,175.620,15.355,152.167
C04825=1096.180,-22.275,-52.696,175.618,15.354,152.167
C04826=1096.175,-22.525,-52.683,175.617,15.353,152.167
C04827=1096.170,-22.775,-52.670,175.615,15.352,152.167
C04828=1096.163,-23.024,-52.657,175.613,15.352,152.167
C04829=1096.157,-23.274,-52.645,175.612,15.350,152.168
C04830=1096.152,-23.524,-52.632,175.610,15.350,152.168
C04831=1096.145,-23.773,-52.619,175.608,15.349,152.168
C04832=1096.140,-24.022,-52.607,175.606,15.348,152.168
C04833=1096.134,-24.272,-52.594,175.604,15.347,152.168
C04834=1096.129,-24.522,-52.581,175.602,15.346,152.169
C04835=1096.123,-24.771,-52.568,175.600,15.345,152.169
C04836=1096.117,-25.021,-52.555,175.598,15.344,152.169
C04837=1096.111,-25.271,-52.543,175.597,15.343,152.169
C04838=1096.105,-25.520,-52.530,175.595,15.342,152.169
C04839=1096.099,-25.770,-52.517,175.593,15.341,152.170
C04840=1096.093,-26.019,-52.505,175.591,15.340,152.170
C04841=1096.088,-26.269,-52.492,175.589,15.339,152.170
C04842=1096.082,-26.519,-52.480,175.588,15.338,152.170
C04843=1096.076,-26.768,-52.467,175.586,15.337,152.170
C04844=1096.070,-27.018,-52.454,175.584,15.337,152.171
C04845=1096.064,-27.268,-52.441,175.582,15.336,152.171
C04846=1096.058,-27.517,-52.429,175.580,15.334,152.171
C04847=1096.052,-27.767,-52.416,175.578,15.334,152.171
C04848=1096.047,-28.016,-52.403,175.576,15.332,152.171
C04849=1096.041,-28.266,-52.391,175.574,15.332,152.172
C04850=1096.035,-28.516,-52.378,175.572,15.331,152.172
C04851=1096.029,-28.766,-52.366,175.571,15.330,152.172
C04852=1096.023,-29.015,-52.353,175.569,15.329,152.172
C04853=1096.018,-29.264,-52.340,175.567,15.328,152.173
C04854=1096.012,-29.514,-52.328,175.566,15.327,152.173
C04855=1096.006,-29.764,-52.315,175.564,15.326,152.173
C04856=1096.000,-30.014,-52.303,175.562,15.326,152.173
C04857=1095.993,-30.263,-52.291,175.560,15.325,152.173
C04858=1095.988,-30.512,-52.278,175.558,15.324,152.173
C04859=1095.982,-30.762,-52.266,175.556,15.323,152.174
C04860=1095.976,-31.012,-52.253,175.555,15.322,152.174
C04861=1095.970,-31.261,-52.240,175.553,15.321,152.174
C04862=1095.965,-31.511,-52.228,175.551,15.319,152.174
C04863=1095.959,-31.760,-52.215,175.549,15.319,152.175
C04864=1095.953,-32.010,-52.203,175.547,15.318,152.175
C04865=1095.946,-32.279,-52.189,175.545,15.317,152.175
C04866=1095.940,-32.547,-52.176,175.543,15.316,152.175
C04867=1095.934,-32.815,-52.162,175.541,15.315,152.175
C04868=1095.927,-33.083,-52.150,175.540,15.315,152.176
C04869=1095.921,-33.332,-52.137,175.538,15.314,152.176
C04870=1095.915,-33.582,-52.125,175.535,15.312,152.176
C04871=1095.910,-33.832,-52.113,175.534,15.311,152.176
C04872=1095.904,-34.081,-52.100,175.532,15.310,152.176
C04873=1095.898,-34.331,-52.087,175.530,15.310,152.177
C04874=1095.892,-34.581,-52.075,175.528,15.308,152.177
C04875=1095.886,-34.830,-52.063,175.527,15.308,152.177
C04876=1095.880,-35.080,-52.051,175.525,15.307,152.177
C04877=1095.874,-35.330,-52.038,175.523,15.306,152.177
C04878=1095.869,-35.579,-52.026,175.521,15.305,152.178
C04879=1095.863,-35.829,-52.013,175.520,15.304,152.178
C04880=1095.857,-36.079,-52.001,175.518,15.303,152.178
C04881=1095.851,-36.328,-51.989,175.516,15.302,152.178
C04882=1095.845,-36.578,-51.977,175.514,15.301,152.178
C04883=1095.839,-36.827,-51.964,175.512,15.301,152.179
C04884=1095.834,-37.077,-51.952,175.511,15.299,152.179
C04885=1095.828,-37.326,-51.939,175.509,15.299,152.179
C04886=1095.822,-37.577,-51.928,175.507,15.298,152.179
C04887=1095.816,-37.826,-51.916,175.505,15.297,152.179
C04888=1095.811,-38.076,-51.904,175.504,15.296,152.180
C04889=1095.805,-38.326,-51.891,175.502,15.295,152.180
C04890=1095.799,-38.575,-51.879,175.500,15.294,152.180
C04891=1095.793,-38.824,-51.867,175.498,15.293,152.180
C04892=1095.787,-39.074,-51.854,175.497,15.292,152.180
C04893=1095.781,-39.323,-51.842,175.495,15.292,152.181
C04894=1095.775,-39.573,-51.830,175.493,15.291,152.181
C04895=1095.769,-39.824,-51.818,175.491,15.290,152.181
C04896=1095.764,-40.073,-51.806,175.489,15.289,152.181
C04897=1095.757,-40.322,-51.794,175.487,15.288,152.181
C04898=1095.751,-40.572,-51.782,175.486,15.287,152.182
C04899=1095.745,-40.822,-51.769,175.484,15.286,152.182
C04900=1095.739,-41.071,-51.757,175.482,15.286,152.182
C04901=1095.733,-41.321,-51.745,175.481,15.284,152.182
C04902=1095.728,-41.570,-51.734,175.479,15.284,152.182
C04903=1095.722,-41.820,-51.721,175.477,15.283,152.183
C04904=1095.716,-42.070,-51.709,175.475,15.282,152.183
C04905=1095.710,-42.319,-51.697,175.473,15.281,152.183
C04906=1095.704,-42.569,-51.685,175.471,15.280,152.183
C04907=1095.698,-42.819,-51.673,175.470,15.279,152.183
C04908=1095.692,-43.068,-51.661,175.468,15.279,152.184
C04909=1095.686,-43.318,-51.649,175.466,15.278,152.184
C04910=1095.680,-43.568,-51.637,175.464,15.277,152.184
C04911=1095.675,-43.817,-51.625,175.463,15.276,152.184
C04912=1095.669,-44.067,-51.613,175.461,15.275,152.185
C04913=1095.663,-44.316,-51.601,175.459,15.274,152.185
C04914=1095.657,-44.566,-51.589,175.457,15.273,152.185
C04915=1095.651,-44.816,-51.577,175.456,15.272,152.185
C04916=1095.645,-45.065,-51.565,175.454,15.271,152.185
C04917=1095.639,-45.315,-51.553,175.452,15.271,152.186
C04918=1095.633,-45.564,-51.541,175.450,15.270,152.186
C04919=1095.628,-45.815,-51.529,175.448,15.269,152.186
C04920=1095.621,-46.064,-51.517,175.447,15.268,152.186
C04921=1095.616,-46.313,-51.505,175.445,15.267,152.186
C04922=1095.609,-46.564,-51.494,175.443,15.266,152.187
C04923=1095.604,-46.813,-51.482,175.441,15.266,152.187
C04924=1095.597,-47.062,-51.470,175.440,15.264,152.187
C04925=1095.592,-47.313,-51.458,175.438,15.264,152.187
C04926=1095.586,-47.562,-51.446,175.436,15.262,152.187
C04927=1095.580,-47.812,-51.434,175.434,15.262,152.188
C04928=1095.575,-48.061,-51.422,175.432,15.261,152.188
C04929=1095.568,-48.330,-51.409,175.431,15.260,152.188
C04930=1095.562,-48.598,-51.397,175.429,15.259,152.188
C04931=1095.556,-48.867,-51.384,175.427,15.258,152.188
C04932=1095.549,-49.136,-51.372,175.425,15.257,152.189
C04933=1095.543,-49.385,-51.359,175.423,15.256,152.189
C04934=1095.537,-49.635,-51.347,175.421,15.255,152.189
C04935=1095.532,-49.884,-51.336,175.419,15.254,152.189
C04936=1095.525,-50.134,-51.324,175.418,15.254,152.189
C04937=1095.520,-50.384,-51.313,175.416,15.253,152.190
C04938=1095.513,-50.633,-51.301,175.415,15.252,152.190
C04939=1095.508,-50.883,-51.289,175.413,15.251,152.190
C04940=1095.502,-51.133,-51.277,175.411,15.251,152.190
C04941=1095.496,-51.382,-51.266,175.409,15.249,152.190
C04942=1095.490,-51.632,-51.254,175.407,15.249,152.191
C04943=1095.484,-51.882,-51.242,175.406,15.248,152.191
C04944=1095.478,-52.131,-51.231,175.404,15.247,152.191
C04945=1095.471,-52.381,-51.219,175.402,15.246,152.191
C04946=1095.466,-52.631,-51.207,175.400,15.245,152.192
C04947=1095.459,-52.880,-51.196,175.398,15.245,152.192
C04948=1095.453,-53.130,-51.184,175.396,15.244,152.192
C04949=1095.448,-53.380,-51.172,175.395,15.243,152.192
C04950=1095.442,-53.630,-51.161,175.393,15.242,152.192
C04951=1095.435,-53.879,-51.149,175.391,15.241,152.193
C04952=1095.429,-54.129,-51.138,175.389,15.241,152.193
C04953=1095.424,-54.378,-51.126,175.388,15.240,152.193
C04954=1095.417,-54.628,-51.115,175.387,15.239,152.193
C04955=1095.411,-54.877,-51.103,175.385,15.239,152.194
C04956=1095.405,-55.127,-51.092,175.383,15.238,152.194
C04957=1095.399,-55.377,-51.079,175.381,15.237,152.194
C04958=1095.393,-55.627,-51.068,175.379,15.236,152.194
C04959=1095.387,-55.876,-51.056,175.377,15.235,152.194
C04960=1095.381,-56.126,-51.045,175.376,15.234,152.195
C04961=1095.375,-56.376,-51.033,175.374,15.234,152.195
C04962=1095.369,-56.625,-51.022,175.372,15.233,152.195
C04963=1095.363,-56.875,-51.011,175.370,15.232,152.195
C04964=1095.357,-57.124,-50.999,175.369,15.231,152.195
C04965=1095.351,-57.375,-50.987,175.367,15.230,152.196
C04966=1095.345,-57.623,-50.976,175.365,15.230,152.196
C04967=1095.339,-57.874,-50.965,175.364,15.229,152.196
C04968=1095.333,-58.123,-50.954,175.362,15.228,152.196
C04969=1095.327,-58.373,-50.941,175.360,15.228,152.197
C04970=1095.322,-58.623,-50.930,175.358,15.227,152.197
C04971=1095.315,-58.873,-50.919,175.357,15.226,152.197
C04972=1095.309,-59.122,-50.907,175.355,15.225,152.197
C04973=1095.304,-59.371,-50.897,175.353,15.224,152.197
C04974=1095.298,-59.621,-50.884,175.351,15.223,152.198
C04975=1095.292,-59.870,-50.873,175.350,15.222,152.198
C04976=1095.286,-60.121,-50.862,175.348,15.222,152.198
C04977=1095.279,-60.370,-50.850,175.346,15.221,152.198
C04978=1095.273,-60.620,-50.839,175.345,15.220,152.198
C04979=1095.268,-60.870,-50.828,175.343,15.220,152.199
C04980=1095.262,-61.120,-50.816,175.341,15.219,152.199
C04981=1095.256,-61.369,-50.805,175.340,15.218,152.199
C04982=1095.249,-61.619,-50.793,175.338,15.217,152.199
C04983=1095.244,-61.868,-50.783,175.336,15.216,152.200
C04984=1095.238,-62.117,-50.771,175.334,15.216,152.200
C04985=1095.232,-62.368,-50.759,175.332,15.215,152.200
C04986=1095.226,-62.617,-50.748,175.330,15.214,152.200
C04987=1095.220,-62.867,-50.737,175.329,15.213,152.200
C04988=1095.214,-63.116,-50.725,175.327,15.213,152.201
C04989=1095.208,-63.366,-50.715,175.326,15.212,152.201
C04990=1095.202,-63.616,-50.703,175.324,15.211,152.201
C04991=1095.196,-63.865,-50.692,175.322,15.210,152.201
C04992=1095.190,-64.115,-50.680,175.321,15.209,152.201
C04993=1095.184,-64.385,-50.669,175.319,15.209,152.202
C04994=1095.178,-64.655,-50.657,175.317,15.208,152.202
C04995=1095.171,-64.925,-50.644,175.315,15.207,152.202
C04996=1095.164,-65.194,-50.632,175.313,15.206,152.202
C04997=1095.159,-65.444,-50.621,175.311,15.205,152.203
C04998=1095.153,-65.694,-50.609,175.310,15.205,152.203
C04999=1095.147,-65.944,-50.599,175.308,15.204,152.203
C05000=1095.141,-66.193,-50.587,175.306,15.203,152.203
C05001=1095.135,-66.443,-50.576,175.304,15.202,152.203
C05002=1095.129,-66.692,-50.565,175.303,15.202,152.204
C05003=1095.123,-66.943,-50.554,175.301,15.201,152.204
C05004=1095.117,-67.192,-50.543,175.300,15.200,152.204
C05005=1095.111,-67.442,-50.532,175.298,15.199,152.204
C05006=1095.106,-67.692,-50.520,175.296,15.199,152.205
C05007=1095.100,-67.941,-50.508,175.294,15.197,152.205
C05008=1095.094,-68.190,-50.498,175.292,15.197,152.205
C05009=1095.088,-68.441,-50.486,175.290,15.196,152.205
C05010=1095.082,-68.690,-50.475,175.289,15.196,152.205
C05011=1095.076,-68.940,-50.465,175.288,15.195,152.205
C05012=1095.070,-69.190,-50.453,175.286,15.194,152.206
C05013=1095.064,-69.439,-50.442,175.284,15.193,152.206
C05014=1095.058,-69.689,-50.432,175.282,15.193,152.206
C05015=1095.053,-69.938,-50.421,175.281,15.191,152.206
C05016=1095.046,-70.188,-50.409,175.279,15.191,152.207
C05017=1095.040,-70.438,-50.399,175.278,15.191,152.207
C05018=1095.035,-70.687,-50.388,175.276,15.189,152.207
C05019=1095.029,-70.938,-50.376,175.274,15.189,152.207
C05020=1095.023,-71.187,-50.365,175.272,15.188,152.208
C05021=1095.018,-71.437,-50.354,175.270,15.187,152.208
C05022=1095.012,-71.686,-50.343,175.269,15.186,152.208
C05023=1095.006,-71.937,-50.332,175.268,15.186,152.208
C05024=1095.000,-72.186,-50.321,175.266,15.185,152.208
C05025=1094.994,-72.436,-50.310,175.264,15.184,152.208
C05026=1094.988,-72.686,-50.299,175.262,15.183,152.209
C05027=1094.982,-72.935,-50.288,175.260,15.183,152.209
C05028=1094.976,-73.185,-50.277,175.258,15.182,152.209
C05029=1094.971,-73.434,-50.266,175.257,15.181,152.209
C05030=1094.965,-73.684,-50.255,175.256,15.181,152.210
C05031=1094.958,-73.934,-50.244,175.254,15.180,152.210
C05032=1094.953,-74.183,-50.233,175.252,15.179,152.210
C05033=1094.947,-74.433,-50.222,175.250,15.178,152.210
C05034=1094.941,-74.683,-50.211,175.249,15.177,152.210
C05035=1094.935,-74.933,-50.200,175.247,15.177,152.211
C05036=1094.928,-75.182,-50.190,175.246,15.177,152.211
C05037=1094.923,-75.431,-50.179,175.244,15.176,152.211
C05038=1094.916,-75.681,-50.168,175.242,15.175,152.211
C05039=1094.911,-75.931,-50.157,175.240,15.174,152.212
C05040=1094.905,-76.180,-50.146,175.238,15.173,152.212
C05041=1094.899,-76.431,-50.135,175.237,15.173,152.212
C05042=1094.893,-76.680,-50.124,175.235,15.173,152.212
C05043=1094.886,-76.929,-50.114,175.233,15.172,152.213
C05044=1094.881,-77.179,-50.104,175.232,15.171,152.213
C05045=1094.875,-77.430,-50.092,175.230,15.170,152.213
C05046=1094.869,-77.679,-50.081,175.229,15.170,152.213
C05047=1094.863,-77.929,-50.071,175.227,15.169,152.213
C05048=1094.857,-78.178,-50.060,175.225,15.168,152.214
C05049=1094.850,-78.428,-50.049,175.223,15.168,152.214
C05050=1094.845,-78.677,-50.038,175.222,15.167,152.214
C05051=1094.839,-78.927,-50.028,175.220,15.167,152.214
C05052=1094.833,-79.177,-50.017,175.219,15.166,152.215
C05053=1094.827,-79.427,-50.006,175.217,15.165,152.215
C05054=1094.821,-79.676,-49.996,175.215,15.164,152.215
C05055=1094.815,-79.926,-49.985,175.213,15.163,152.215
C05056=1094.809,-80.175,-49.974,175.212,15.163,152.215
C05057=1094.803,-80.448,-49.963,175.210,15.162,152.216
C05058=1094.796,-80.720,-49.951,175.208,15.162,152.216
C05059=1094.789,-80.992,-49.939,175.206,15.161,152.216
C05060=1094.782,-81.264,-49.928,175.205,15.160,152.217
C05061=1094.776,-81.514,-49.917,175.203,15.160,152.217
C05062=1094.770,-81.763,-49.906,175.201,15.159,152.217
C05063=1094.763,-82.013,-49.896,175.199,15.158,152.217
C05064=1094.758,-82.263,-49.885,175.198,15.158,152.218
C05065=1094.752,-82.513,-49.875,175.196,15.157,152.218
C05066=1094.746,-82.762,-49.864,175.194,15.157,152.218
C05067=1094.739,-83.012,-49.853,175.192,15.156,152.218
C05068=1094.734,-83.262,-49.843,175.191,15.156,152.219
C05069=1094.727,-83.511,-49.833,175.189,15.155,152.219
C05070=1094.722,-83.761,-49.822,175.188,15.154,152.219
C05071=1094.715,-84.010,-49.811,175.186,15.153,152.219
C05072=1094.709,-84.261,-49.801,175.184,15.153,152.219
C05073=1094.703,-84.510,-49.790,175.183,15.153,152.220
C05074=1094.697,-84.759,-49.780,175.181,15.152,152.220
C05075=1094.692,-85.009,-49.770,175.179,15.151,152.220
C05076=1094.685,-85.260,-49.758,175.177,15.151,152.220
C05077=1094.679,-85.509,-49.748,175.176,15.150,152.221
C05078=1094.673,-85.758,-49.737,175.174,15.150,152.221
C05079=1094.667,-86.008,-49.728,175.172,15.149,152.221
C05080=1094.661,-86.258,-49.717,175.170,15.148,152.221
C05081=1094.655,-86.508,-49.705,175.169,15.148,152.222
C05082=1094.649,-86.758,-49.696,175.168,15.147,152.222
C05083=1094.643,-87.007,-49.685,175.166,15.146,152.222
C05084=1094.637,-87.257,-49.675,175.164,15.146,152.222
C05085=1094.631,-87.506,-49.665,175.163,15.146,152.223
C05086=1094.624,-87.756,-49.654,175.161,15.145,152.223
C05087=1094.618,-88.006,-49.644,175.159,15.144,152.223
C05088=1094.613,-88.256,-49.633,175.157,15.143,152.223
C05089=1094.606,-88.505,-49.623,175.156,15.143,152.224
C05090=1094.601,-88.755,-49.612,175.154,15.143,152.224
C05091=1094.594,-89.004,-49.602,175.152,15.142,152.224
C05092=1094.589,-89.254,-49.592,175.150,15.141,152.224
C05093=1094.582,-89.504,-49.581,175.149,15.141,152.225
C05094=1094.576,-89.754,-49.570,175.147,15.140,152.225
C05095=1094.571,-90.004,-49.560,175.146,15.139,152.225
C05096=1094.564,-90.253,-49.550,175.144,15.139,152.225
C05097=1094.559,-90.503,-49.540,175.143,15.139,152.225
C05098=1094.552,-90.752,-49.530,175.141,15.138,152.226
C05099=1094.547,-91.002,-49.519,175.139,15.137,152.226
C05100=1094.540,-91.252,-49.509,175.138,15.137,152.226
C05101=1094.534,-91.502,-49.498,175.136,15.136,152.226
C05102=1094.528,-91.752,-49.488,175.134,15.136,152.227
C05103=1094.522,-92.001,-49.477,175.132,15.135,152.227
C05104=1094.516,-92.251,-49.468,175.131,15.135,152.227
C05105=1094.510,-92.500,-49.457,175.129,15.134,152.228
C05106=1094.504,-92.750,-49.447,175.127,15.133,152.228
C05107=1094.498,-93.000,-49.437,175.126,15.133,152.228
C05108=1094.492,-93.249,-49.427,175.124,15.133,152.228
C05109=1094.486,-93.499,-49.416,175.122,15.132,152.229
C05110=1094.480,-93.749,-49.407,175.120,15.131,152.229
C05111=1094.474,-93.999,-49.395,175.119,15.131,152.229
C05112=1094.468,-94.249,-49.386,175.117,15.131,152.229
C05113=1094.462,-94.498,-49.375,175.115,15.130,152.230
C05114=1094.456,-94.748,-49.365,175.114,15.130,152.230
C05115=1094.450,-94.998,-49.355,175.113,15.129,152.230
C05116=1094.444,-95.247,-49.345,175.111,15.128,152.230
C05117=1094.438,-95.497,-49.335,175.109,15.127,152.230
C05118=1094.432,-95.747,-49.324,175.108,15.127,152.231
C05119=1094.426,-95.997,-49.314,175.106,15.126,152.231
C05120=1094.420,-96.246,-49.304,175.104,15.126,152.231
C05121=1094.414,-96.520,-49.292,175.102,15.125,152.231
C05122=1094.407,-96.795,-49.282,175.101,15.125,152.232
C05123=1094.401,-97.070,-49.270,175.099,15.125,152.232
C05124=1094.394,-97.344,-49.260,175.097,15.124,152.232
C05125=1094.388,-97.593,-49.249,175.095,15.123,152.233
C05126=1094.382,-97.843,-49.239,175.094,15.123,152.233
C05127=1094.376,-98.093,-49.229,175.092,15.123,152.233
C05128=1094.370,-98.342,-49.219,175.090,15.122,152.233
C05129=1094.364,-98.592,-49.209,175.088,15.121,152.234
C05130=1094.357,-98.842,-49.199,175.087,15.121,152.234
C05131=1094.351,-99.092,-49.189,175.085,15.120,152.234
C05132=1094.346,-99.342,-49.179,175.083,15.120,152.234
C05133=1094.339,-99.591,-49.168,175.082,15.120,152.235
C05134=1094.333,-99.841,-49.159,175.080,15.119,152.235
C05135=1094.327,-100.091,-49.149,175.079,15.118,152.235
C05136=1094.321,-100.340,-49.138,175.077,15.118,152.235
C05137=1094.315,-100.590,-49.129,175.076,15.117,152.236
C05138=1094.309,-100.840,-49.119,175.074,15.117,152.236
C05139=1094.303,-101.089,-49.108,175.073,15.117,152.236
C05140=1094.297,-101.339,-49.099,175.071,15.116,152.236
C05141=1094.291,-101.589,-49.089,175.068,15.116,152.237
C05142=1094.285,-101.839,-49.079,175.067,15.116,152.237
C05143=1094.279,-102.088,-49.069,175.065,15.115,152.237
C05144=1094.272,-102.338,-49.059,175.064,15.114,152.238
C05145=1094.266,-102.588,-49.050,175.062,15.114,152.238
C05146=1094.261,-102.837,-49.039,175.061,15.113,152.238
C05147=1094.254,-103.087,-49.029,175.059,15.113,152.238
C05148=1094.248,-103.337,-49.020,175.058,15.113,152.239
C05149=1094.243,-103.587,-49.009,175.056,15.112,152.239
C05150=1094.236,-103.836,-48.999,175.055,15.112,152.239
C05151=1094.230,-104.086,-48.990,175.053,15.111,152.239
C05152=1094.224,-104.336,-48.980,175.050,15.111,152.240
C05153=1094.218,-104.585,-48.970,175.049,15.111,152.240
C05154=1094.212,-104.835,-48.960,175.047,15.110,152.240
C05155=1094.206,-105.085,-48.950,175.046,15.110,152.241
C05156=1094.200,-105.334,-48.940,175.044,15.109,152.241
C05157=1094.194,-105.584,-48.931,175.043,15.109,152.241
C05158=1094.188,-105.834,-48.920,175.041,15.108,152.241
C05159=1094.182,-106.083,-48.910,175.040,15.108,152.242
C05160=1094.175,-106.333,-48.901,175.038,15.107,152.242
C05161=1094.169,-106.583,-48.891,175.035,15.107,152.242
C05162=1094.163,-106.833,-48.882,175.034,15.107,152.242
C05163=1094.158,-107.083,-48.872,175.032,15.106,152.243
C05164=1094.151,-107.332,-48.861,175.031,15.106,152.243
C05165=1094.145,-107.582,-48.852,175.029,15.105,152.243
C05166=1094.139,-107.832,-48.842,175.028,15.105,152.243
C05167=1094.133,-108.082,-48.833,175.026,15.105,152.244
C05168=1094.127,-108.331,-48.823,175.024,15.105,152.244
C05169=1094.120,-108.581,-48.813,175.022,15.104,152.244
C05170=1094.115,-108.831,-48.803,175.021,15.104,152.245
C05171=1094.108,-109.080,-48.793,175.019,15.103,152.245
C05172=1094.102,-109.330,-48.783,175.018,15.103,152.245
C05173=1094.096,-109.580,-48.774,175.016,15.102,152.245
C05174=1094.090,-109.830,-48.764,175.014,15.102,152.246
C05175=1094.084,-110.080,-48.755,175.013,15.102,152.246
C05176=1094.078,-110.329,-48.745,175.011,15.101,152.246
C05177=1094.071,-110.579,-48.736,175.010,15.101,152.247
C05178=1094.065,-110.828,-48.725,175.008,15.101,152.247
C05179=1094.059,-111.078,-48.716,175.006,15.100,152.247
C05180=1094.053,-111.328,-48.706,175.005,15.100,152.247
C05181=1094.046,-111.578,-48.697,175.003,15.100,152.248
C05182=1094.041,-111.828,-48.686,175.002,15.099,152.248
C05183=1094.035,-112.078,-48.677,175.000,15.099,152.248
C05184=1094.029,-112.328,-48.667,174.998,15.099,152.249
C05185=1094.022,-112.592,-48.657,174.997,15.098,152.249
C05186=1094.016,-112.859,-48.647,174.995,15.098,152.249
C05187=1094.009,-113.124,-48.637,174.993,15.097,152.249
C05188=1094.002,-113.390,-48.627,174.991,15.098,152.250
C05189=1093.996,-113.639,-48.617,174.990,15.097,152.250
C05190=1093.990,-113.889,-48.608,174.988,15.096,152.250
C05191=1093.984,-114.138,-48.598,174.987,15.096,152.251
C05192=1093.978,-114.388,-48.589,174.985,15.095,152.251
C05193=1093.972,-114.638,-48.579,174.983,15.096,152.251
C05194=1093.966,-114.888,-48.569,174.981,15.095,152.251
C05195=1093.959,-115.138,-48.560,174.979,15.094,152.252
C05196=1093.953,-115.387,-48.550,174.978,15.094,152.252
C05197=1093.947,-115.637,-48.541,174.976,15.094,152.252
C05198=1093.941,-115.887,-48.531,174.975,15.094,152.253
C05199=1093.935,-116.137,-48.522,174.973,15.093,152.253
C05200=1093.928,-116.387,-48.512,174.972,15.093,152.253
C05201=1093.923,-116.636,-48.504,174.970,15.093,152.254
C05202=1093.917,-116.886,-48.494,174.968,15.092,152.254
C05203=1093.911,-117.136,-48.484,174.967,15.092,152.254
C05204=1093.905,-117.386,-48.475,174.965,15.092,152.254
C05205=1093.899,-117.635,-48.465,174.963,15.092,152.255
C05206=1093.892,-117.885,-48.456,174.962,15.091,152.255
C05207=1093.886,-118.135,-48.446,174.960,15.091,152.255
C05208=1093.880,-118.385,-48.437,174.958,15.091,152.256
C05209=1093.874,-118.635,-48.427,174.956,15.090,152.256
C05210=1093.868,-118.884,-48.417,174.955,15.090,152.256
C05211=1093.862,-119.134,-48.408,174.953,15.090,152.257
C05212=1093.855,-119.383,-48.399,174.952,15.090,152.257
C05213=1093.849,-119.633,-48.390,174.950,15.089,152.257
C05214=1093.843,-119.883,-48.380,174.949,15.089,152.257
C05215=1093.837,-120.133,-48.371,174.947,15.089,152.258
C05216=1093.831,-120.383,-48.362,174.946,15.089,152.258
C05217=1093.825,-120.633,-48.352,174.944,15.088,152.258
C05218=1093.818,-120.882,-48.343,174.942,15.088,152.259
C05219=1093.813,-121.132,-48.333,174.940,15.088,152.259
C05220=1093.807,-121.381,-48.324,174.939,15.087,152.259
C05221=1093.800,-121.631,-48.315,174.937,15.088,152.260
C05222=1093.794,-121.881,-48.306,174.935,15.087,152.260
C05223=1093.788,-122.131,-48.296,174.934,15.087,152.260
C05224=1093.782,-122.381,-48.287,174.932,15.087,152.260
C05225=1093.775,-122.631,-48.277,174.931,15.087,152.261
C05226=1093.770,-122.880,-48.268,174.929,15.086,152.261
C05227=1093.763,-123.129,-48.259,174.927,15.086,152.261
C05228=1093.757,-123.380,-48.250,174.926,15.086,152.262
C05229=1093.751,-123.629,-48.241,174.924,15.086,152.262
C05230=1093.745,-123.879,-48.231,174.922,15.085,152.262
C05231=1093.739,-124.129,-48.222,174.920,15.085,152.263
C05232=1093.733,-124.378,-48.212,174.919,15.085,152.263
C05233=1093.726,-124.628,-48.204,174.917,15.084,152.263
C05234=1093.720,-124.878,-48.195,174.916,15.084,152.263
C05235=1093.714,-125.128,-48.185,174.914,15.084,152.264
C05236=1093.708,-125.378,-48.175,174.913,15.084,152.264
C05237=1093.702,-125.627,-48.166,174.911,15.083,152.264
C05238=1093.695,-125.878,-48.158,174.909,15.084,152.265
C05239=1093.690,-126.127,-48.148,174.907,15.083,152.265
C05240=1093.683,-126.376,-48.139,174.906,15.083,152.265
C05241=1093.676,-126.626,-48.130,174.904,15.083,152.266
C05242=1093.671,-126.876,-48.121,174.903,15.083,152.266
C05243=1093.664,-127.126,-48.111,174.901,15.083,152.266
C05244=1093.659,-127.375,-48.102,174.900,15.082,152.267
C05245=1093.652,-127.636,-48.093,174.897,15.082,152.267
C05246=1093.645,-127.896,-48.083,174.896,15.082,152.267
C05247=1093.639,-128.156,-48.074,174.894,15.081,152.267
C05248=1093.642,-128.415,-48.061,174.894,15.079,152.267
C05249=1093.235,-128.436,-48.176,174.849,15.187,152.298
C05250=1093.232,-128.178,-48.188,174.849,15.191,152.298
C05251=1093.238,-127.917,-48.198,174.851,15.191,152.298
C05252=1093.244,-127.658,-48.207,174.853,15.192,152.297
C05253=1093.250,-127.398,-48.216,174.854,15.192,152.297
C05254=1093.256,-127.148,-48.226,174.857,15.192,152.297
C05255=1093.263,-126.898,-48.235,174.858,15.192,152.297
C05256=1093.269,-126.649,-48.244,174.860,15.192,152.296
C05257=1093.275,-126.398,-48.253,174.861,15.192,152.296
C05258=1093.281,-126.149,-48.263,174.863,15.193,152.296
C05259=1093.288,-125.900,-48.271,174.864,15.192,152.295
C05260=1093.294,-125.650,-48.281,174.866,15.193,152.295
C05261=1093.300,-125.399,-48.290,174.867,15.193,152.295
C05262=1093.306,-125.150,-48.299,174.870,15.193,152.294
C05263=1093.313,-124.900,-48.308,174.871,15.193,152.294
C05264=1093.319,-124.650,-48.318,174.873,15.194,152.294
C05265=1093.324,-124.401,-48.327,174.874,15.194,152.293
C05266=1093.330,-124.151,-48.336,174.876,15.194,152.293
C05267=1093.337,-123.901,-48.346,174.878,15.195,152.293
C05268=1093.344,-123.651,-48.355,174.879,15.195,152.293
C05269=1093.350,-123.402,-48.364,174.881,15.195,152.292
C05270=1093.356,-123.151,-48.373,174.882,15.195,152.292
C05271=1093.361,-122.902,-48.382,174.884,15.196,152.292
C05272=1093.367,-122.652,-48.392,174.886,15.196,152.291
C05273=1093.373,-122.403,-48.401,174.887,15.196,152.291
C05274=1093.380,-122.153,-48.410,174.889,15.196,152.291
C05275=1093.387,-121.903,-48.420,174.891,15.197,152.290
C05276=1093.392,-121.653,-48.429,174.892,15.197,152.290
C05277=1093.398,-121.404,-48.438,174.894,15.197,152.290
C05278=1093.404,-121.154,-48.448,174.896,15.198,152.290
C05279=1093.410,-120.904,-48.457,174.897,15.198,152.289
C05280=1093.416,-120.654,-48.467,174.899,15.198,152.289
C05281=1093.423,-120.405,-48.476,174.900,15.198,152.289
C05282=1093.430,-120.155,-48.485,174.902,15.199,152.288
C05283=1093.435,-119.905,-48.494,174.903,15.199,152.288
C05284=1093.442,-119.655,-48.504,174.905,15.199,152.288
C05285=1093.447,-119.406,-48.513,174.907,15.200,152.288
C05286=1093.453,-119.156,-48.522,174.909,15.200,152.287
C05287=1093.460,-118.906,-48.532,174.910,15.200,152.287
C05288=1093.466,-118.656,-48.542,174.912,15.200,152.287
C05289=1093.472,-118.407,-48.551,174.913,15.201,152.286
C05290=1093.478,-118.157,-48.561,174.915,15.201,152.286
C05291=1093.484,-117.907,-48.570,174.917,15.201,152.286
C05292=1093.490,-117.657,-48.580,174.918,15.201,152.286
C05293=1093.497,-117.408,-48.589,174.920,15.202,152.285
C05294=1093.503,-117.159,-48.598,174.922,15.202,152.285
C05295=1093.509,-116.909,-48.608,174.923,15.202,152.285
C05296=1093.515,-116.658,-48.616,174.925,15.203,152.284
C05297=1093.521,-116.409,-48.626,174.926,15.203,152.284
C05298=1093.527,-116.159,-48.636,174.928,15.204,152.284
C05299=1093.533,-115.909,-48.645,174.930,15.204,152.283
C05300=1093.540,-115.659,-48.655,174.931,15.204,152.283
C05301=1093.546,-115.409,-48.664,174.933,15.205,152.283
C05302=1093.552,-115.160,-48.674,174.934,15.205,152.283
C05303=1093.558,-114.910,-48.683,174.937,15.205,152.282
C05304=1093.564,-114.660,-48.693,174.938,15.205,152.282
C05305=1093.570,-114.410,-48.702,174.940,15.206,152.282
C05306=1093.576,-114.161,-48.712,174.941,15.206,152.282
C05307=1093.582,-113.911,-48.721,174.943,15.207,152.281
C05308=1093.588,-113.662,-48.731,174.944,15.207,152.281
C05309=1093.595,-113.412,-48.740,174.946,15.207,152.281
C05310=1093.601,-113.146,-48.751,174.948,15.208,152.280
C05311=1093.607,-112.880,-48.761,174.950,15.208,152.280
C05312=1093.614,-112.614,-48.772,174.952,15.209,152.280
C05313=1093.621,-112.348,-48.782,174.953,15.208,152.279
C05314=1093.627,-112.098,-48.791,174.955,15.209,152.279
C05315=1093.633,-111.848,-48.801,174.957,15.210,152.279
C05316=1093.639,-111.598,-48.811,174.958,15.210,152.279
C05317=1093.645,-111.348,-48.820,174.960,15.211,152.278
C05318=1093.651,-111.099,-48.830,174.961,15.211,152.278
C05319=1093.657,-110.849,-48.840,174.963,15.211,152.278
C05320=1093.663,-110.599,-48.849,174.965,15.212,152.278
C05321=1093.670,-110.350,-48.859,174.966,15.212,152.277
C05322=1093.676,-110.100,-48.869,174.968,15.212,152.277
C05323=1093.682,-109.850,-48.879,174.969,15.212,152.277
C05324=1093.688,-109.600,-48.888,174.971,15.213,152.277
C05325=1093.694,-109.351,-48.898,174.973,15.214,152.276
C05326=1093.701,-109.101,-48.907,174.974,15.214,152.276
C05327=1093.707,-108.851,-48.917,174.976,15.215,152.276
C05328=1093.712,-108.601,-48.927,174.978,15.215,152.275
C05329=1093.719,-108.352,-48.937,174.979,15.215,152.275
C05330=1093.725,-108.102,-48.947,174.981,15.216,152.275
C05331=1093.731,-107.852,-48.956,174.982,15.216,152.275
C05332=1093.737,-107.602,-48.966,174.984,15.216,152.274
C05333=1093.743,-107.353,-48.976,174.986,15.217,152.274
C05334=1093.749,-107.103,-48.985,174.987,15.217,152.274
C05335=1093.755,-106.853,-48.996,174.989,15.218,152.274
C05336=1093.761,-106.603,-49.006,174.991,15.218,152.273
C05337=1093.768,-106.354,-49.015,174.992,15.219,152.273
C05338=1093.774,-106.104,-49.025,174.994,15.219,152.273
C05339=1093.780,-105.854,-49.034,174.996,15.219,152.272
C05340=1093.785,-105.605,-49.045,174.997,15.219,152.272
C05341=1093.791,-105.356,-49.054,174.999,15.220,152.272
C05342=1093.797,-105.106,-49.064,175.001,15.221,152.272
C05343=1093.804,-104.856,-49.073,175.002,15.221,152.271
C05344=1093.809,-104.606,-49.084,175.004,15.222,152.271
C05345=1093.815,-104.357,-49.094,175.005,15.222,152.271
C05346=1093.822,-104.107,-49.103,175.007,15.222,152.271
C05347=1093.828,-103.857,-49.113,175.009,15.223,152.270
C05348=1093.834,-103.607,-49.123,175.010,15.223,152.270
C05349=1093.840,-103.357,-49.134,175.012,15.224,152.270
C05350=1093.847,-103.107,-49.143,175.014,15.225,152.270
C05351=1093.853,-102.857,-49.153,175.015,15.225,152.269
C05352=1093.858,-102.607,-49.163,175.017,15.225,152.269
C05353=1093.865,-102.358,-49.173,175.019,15.226,152.269
C05354=1093.871,-102.108,-49.183,175.020,15.226,152.269
C05355=1093.877,-101.859,-49.193,175.022,15.227,152.268
C05356=1093.883,-101.609,-49.203,175.024,15.227,152.268
C05357=1093.889,-101.359,-49.213,175.025,15.228,152.268
C05358=1093.895,-101.109,-49.223,175.027,15.228,152.268
C05359=1093.901,-100.860,-49.233,175.028,15.229,152.267
C05360=1093.907,-100.610,-49.243,175.030,15.229,152.267
C05361=1093.913,-100.360,-49.253,175.031,15.230,152.267
C05362=1093.920,-100.111,-49.263,175.033,15.230,152.267
C05363=1093.925,-99.861,-49.273,175.036,15.231,152.266
C05364=1093.931,-99.611,-49.283,175.037,15.231,152.266
C05365=1093.938,-99.362,-49.293,175.039,15.231,152.266
C05366=1093.943,-99.112,-49.303,175.040,15.232,152.265
C05367=1093.949,-98.862,-49.313,175.042,15.232,152.265
C05368=1093.956,-98.613,-49.323,175.043,15.233,152.265
C05369=1093.962,-98.363,-49.332,175.045,15.233,152.265
C05370=1093.968,-98.112,-49.343,175.046,15.234,152.264
C05371=1093.974,-97.863,-49.353,175.048,15.234,152.264
C05372=1093.981,-97.613,-49.363,175.050,15.235,152.264
C05373=1093.986,-97.364,-49.374,175.051,15.236,152.264
C05374=1093.993,-97.089,-49.384,175.053,15.236,152.264
C05375=1093.999,-96.815,-49.395,175.055,15.237,152.263
C05376=1094.006,-96.541,-49.407,175.057,15.237,152.263
C05377=1094.012,-96.266,-49.418,175.059,15.238,152.263
C05378=1094.018,-96.017,-49.428,175.060,15.239,152.263
C05379=1094.024,-95.767,-49.439,175.062,15.239,152.262
C05380=1094.030,-95.517,-49.448,175.063,15.240,152.262
C05381=1094.036,-95.267,-49.458,175.065,15.240,152.262
C05382=1094.042,-95.018,-49.469,175.066,15.241,152.262
C05383=1094.048,-94.767,-49.479,175.068,15.241,152.261
C05384=1094.055,-94.518,-49.489,175.070,15.242,152.261
C05385=1094.060,-94.268,-49.500,175.072,15.243,152.261
C05386=1094.067,-94.019,-49.510,175.073,15.243,152.261
C05387=1094.072,-93.769,-49.520,175.075,15.243,152.260
C05388=1094.078,-93.519,-49.530,175.077,15.244,152.260
C05389=1094.084,-93.269,-49.541,175.078,15.245,152.260
C05390=1094.090,-93.020,-49.551,175.080,15.245,152.260
C05391=1094.096,-92.770,-49.561,175.082,15.246,152.259
C05392=1094.102,-92.521,-49.571,175.084,15.247,152.259
C05393=1094.108,-92.271,-49.581,175.085,15.247,152.259
C05394=1094.114,-92.022,-49.592,175.087,15.247,152.259
C05395=1094.120,-91.771,-49.602,175.088,15.248,152.258
C05396=1094.127,-91.522,-49.612,175.090,15.249,152.258
C05397=1094.132,-91.271,-49.623,175.091,15.249,152.258
C05398=1094.139,-91.022,-49.633,175.093,15.250,152.258
C05399=1094.144,-90.772,-49.643,175.095,15.251,152.258
C05400=1094.150,-90.523,-49.653,175.097,15.251,152.257
C05401=1094.156,-90.273,-49.664,175.098,15.252,152.257
C05402=1094.162,-90.023,-49.674,175.100,15.252,152.257
C05403=1094.169,-89.773,-49.685,175.102,15.253,152.257
C05404=1094.174,-89.523,-49.695,175.103,15.253,152.256
C05405=1094.181,-89.274,-49.706,175.105,15.254,152.256
C05406=1094.186,-89.025,-49.716,175.107,15.254,152.256
C05407=1094.193,-88.775,-49.726,175.108,15.256,152.256
C05408=1094.198,-88.525,-49.737,175.109,15.256,152.255
C05409=1094.204,-88.276,-49.746,175.111,15.256,152.255
C05410=1094.211,-88.025,-49.758,175.113,15.257,152.255
C05411=1094.217,-87.776,-49.769,175.115,15.258,152.255
C05412=1094.223,-87.526,-49.778,175.116,15.258,152.254
C05413=1094.228,-87.277,-49.789,175.118,15.259,152.254
C05414=1094.235,-87.027,-49.799,175.120,15.259,152.254
C05415=1094.241,-86.777,-49.810,175.121,15.260,152.254
C05416=1094.247,-86.527,-49.821,175.123,15.261,152.253
C05417=1094.253,-86.277,-49.830,175.124,15.261,152.253
C05418=1094.259,-86.028,-49.841,175.126,15.262,152.253
C05419=1094.265,-85.779,-49.851,175.128,15.263,152.253
C05420=1094.271,-85.528,-49.863,175.130,15.263,152.252
C05421=1094.277,-85.278,-49.873,175.131,15.263,152.252
C05422=1094.283,-85.029,-49.883,175.133,15.265,152.252
C05423=1094.289,-84.780,-49.894,175.135,15.265,152.252
C05424=1094.295,-84.530,-49.904,175.137,15.266,152.252
C05425=1094.302,-84.280,-49.915,175.138,15.266,152.251
C05426=1094.307,-84.030,-49.926,175.140,15.267,152.251
C05427=1094.314,-83.780,-49.935,175.141,15.267,152.251
C05428=1094.319,-83.531,-49.946,175.143,15.268,152.251
C05429=1094.326,-83.282,-49.956,175.145,15.269,152.250
C05430=1094.332,-83.032,-49.968,175.146,15.269,152.250
C05431=1094.338,-82.781,-49.978,175.148,15.270,152.250
C05432=1094.344,-82.532,-49.988,175.150,15.271,152.250
C05433=1094.350,-82.283,-49.999,175.152,15.271,152.249
C05434=1094.356,-82.033,-50.010,175.153,15.272,152.249
C05435=1094.363,-81.783,-50.020,175.155,15.272,152.249
C05436=1094.368,-81.533,-50.031,175.156,15.273,152.249
C05437=1094.374,-81.283,-50.042,175.158,15.274,152.249
C05438=1094.380,-81.012,-50.053,175.160,15.275,152.248
C05439=1094.388,-80.740,-50.064,175.162,15.275,152.248
